LIN {X 0,Y 367.655,Z 436.574,A -85,B 0,C 180,E1 -12880.464,E2 -12880.464} C_VEL
LIN {X 0,Y 367.47,Z 439.697,A -85,B 0,C 180,E1 -12882.738,E2 -12882.738} C_VEL
LIN {X 0,Y 367.357,Z 440.888,A -85,B 0,C 180,E1 -12884.402,E2 -12884.402} C_VEL
LIN {X 0,Y 367.359,Z 441.192,A -85,B 0,C 180,E1 -12885.536,E2 -12885.536} C_VEL
LIN {X 0,Y 367.414,Z 440.944,A -85,B 0,C 180,E1 -12886.98,E2 -12886.98} C_VEL
LIN {X 0,Y 367.622,Z 439.55,A -85,B 0,C 180,E1 -12888.919,E2 -12888.919} C_VEL
LIN {X 0,Y 367.118,Z 438.651,A -85,B 0,C 180,E1 -12889.827,E2 -12889.827} C_VEL
LIN {X 0,Y 364.548,Z 436.647,A -85,B 0,C 180,E1 -12891.296,E2 -12891.296} C_VEL
LIN {X 0,Y 362.068,Z 433.845,A -85,B 0,C 180,E1 -12892.751,E2 -12892.751} C_VEL
LIN {X 0,Y 361.716,Z 431.694,A -85,B 0,C 180,E1 -12893.624,E2 -12893.624} C_VEL
LIN {X 0,Y 362.559,Z 425.865,A -85,B 0,C 180,E1 -12895.55,E2 -12895.55} C_VEL
LIN {X 0,Y 363.427,Z 419.541,A -85,B 0,C 180,E1 -12897.184,E2 -12897.184} C_VEL
LIN {X 0,Y 364.552,Z 411.694,A -85,B 0,C 180,E1 -12898.813,E2 -12898.813} C_VEL
LIN {X 0,Y 365.704,Z 403.264,A -85,B 0,C 180,E1 -12900.234,E2 -12900.234} C_VEL
LIN {X 0,Y 366.982,Z 393.098,A -85,B 0,C 180,E1 -12901.617,E2 -12901.617} C_VEL
LIN {X 0,Y 368.262,Z 382.466,A -85,B 0,C 180,E1 -12902.766,E2 -12902.766} C_VEL
LIN {X 0,Y 369.192,Z 372.107,A -85,B 0,C 180,E1 -12903.67,E2 -12903.67} C_VEL
LIN {X 0,Y 370.135,Z 360.17,A -85,B 0,C 180,E1 -12904.475,E2 -12904.475} C_VEL
LIN {X 0,Y 370.867,Z 347.614,A -85,B 0,C 180,E1 -12905.082,E2 -12905.082} C_VEL
LIN {X 0,Y 371.289,Z 334.414,A -85,B 0,C 180,E1 -12905.493,E2 -12905.493} C_VEL
LIN {X 0,Y 372.995,Z 256.748,A -85,B 0,C 180,E1 -12907.02,E2 -12907.02} C_VEL
LIN {X 0,Y 371.362,Z 249.513,A -85,B 0,C 180,E1 -12907.298,E2 -12907.298} C_VEL
LIN {X 0,Y 364.262,Z 233.198,A -85,B 0,C 180,E1 -12908.217,E2 -12908.217} C_VEL
LIN {X 0,Y 363.464,Z 231.172,A -85,B 0,C 180,E1 -12908.333,E2 -12908.333} C_VEL
LIN {X 0,Y 361.902,Z 224.409,A -85,B 0,C 180,E1 -12910.291,E2 -12910.291} C_VEL
LIN {X 0,Y 361.922,Z 224.406,A -85,B 0,C 180,E1 -12914.35,E2 -12914.35} C_VEL
LIN {X 0,Y 361.875,Z 224.407,A -85,B 0,C 180,E1 -12917.558,E2 -12917.558} C_VEL
LIN {X 0,Y 361.861,Z 224.41,A -85,B 0,C 180,E1 -12920.972,E2 -12920.972} C_VEL
LIN {X 0,Y 361.86,Z 224.405,A -85,B 0,C 180,E1 -12924.654,E2 -12924.654} C_VEL
LIN {X 0,Y 361.822,Z 224.409,A -85,B 0,C 180,E1 -12928.369,E2 -12928.369} C_VEL
LIN {X 0,Y 361.885,Z 224.401,A -85,B 0,C 180,E1 -12930.954,E2 -12930.954} C_VEL
LIN {X 0,Y 361.936,Z 224.399,A -85,B 0,C 180,E1 -12933.474,E2 -12933.474} C_VEL
LIN {X 0,Y 361.884,Z 224.404,A -85,B 0,C 180,E1 -12937.145,E2 -12937.145} C_VEL
LIN {X 0,Y 361.907,Z 224.401,A -85,B 0,C 180,E1 -12940.724,E2 -12940.724} C_VEL
LIN {X 0,Y 361.925,Z 224.4,A -85,B 0,C 180,E1 -12944.226,E2 -12944.226} C_VEL
LIN {X 0,Y 361.977,Z 224.391,A -85,B 0,C 180,E1 -12946.527,E2 -12946.527} C_VEL
LIN {X 0,Y 362.008,Z 224.39,A -85,B 0,C 180,E1 -12949.938,E2 -12949.938} C_VEL
LIN {X 0,Y 362.142,Z 224.371,A -85,B 0,C 180,E1 -12953.314,E2 -12953.314} C_VEL
LIN {X 0,Y 362.254,Z 224.357,A -85,B 0,C 180,E1 -12957.777,E2 -12957.777} C_VEL
LIN {X 0,Y 362.381,Z 224.336,A -85,B 0,C 180,E1 -12960,E2 -12960} C_VEL
LIN {X 0,Y 362.254,Z 224.351,A -85,B 0,C 180,E1 -12962.224,E2 -12962.224} C_VEL
LIN {X 0,Y 362.116,Z 224.367,A -85,B 0,C 180,E1 -12966.688,E2 -12966.688} C_VEL
LIN {X 0,Y 361.98,Z 224.382,A -85,B 0,C 180,E1 -12970.064,E2 -12970.064} C_VEL
LIN {X 0,Y 361.979,Z 224.387,A -85,B 0,C 180,E1 -12973.899,E2 -12973.899} C_VEL
LIN {X 0,Y 361.909,Z 224.405,A -85,B 0,C 180,E1 -12976.936,E2 -12976.936} C_VEL
LIN {X 0,Y 361.856,Z 224.406,A -85,B 0,C 180,E1 -12980.463,E2 -12980.463} C_VEL
LIN {X 0,Y 361.878,Z 224.402,A -85,B 0,C 180,E1 -12984.114,E2 -12984.114} C_VEL
LIN {X 0,Y 361.826,Z 224.408,A -85,B 0,C 180,E1 -12987.786,E2 -12987.786} C_VEL
LIN {X 0,Y 361.812,Z 224.411,A -85,B 0,C 180,E1 -12991.281,E2 -12991.281} C_VEL
LIN {X 0,Y 361.837,Z 224.41,A -85,B 0,C 180,E1 -12994.283,E2 -12994.283} C_VEL
LIN {X 0,Y 361.846,Z 224.407,A -85,B 0,C 180,E1 -12997.223,E2 -12997.223} C_VEL
LIN {X 0,Y 361.82,Z 224.405,A -85,B 0,C 180,E1 -13000.756,E2 -13000.756} C_VEL
LIN {X 0,Y 361.808,Z 224.419,A -85,B 0,C 180,E1 -13004.37,E2 -13004.37} C_VEL
LIN {X 0,Y 361.824,Z 224.413,A -85,B 0,C 180,E1 -13007.571,E2 -13007.571} C_VEL
LIN {X 0,Y 361.838,Z 224.414,A -85,B 0,C 180,E1 -13011.573,E2 -13011.573} C_VEL
LIN {X 0,Y 361.871,Z 224.411,A -85,B 0,C 180,E1 -13014.657,E2 -13014.657} C_VEL
LIN {X 0,Y 361.893,Z 224.531,A -85,B 0,C 180,E1 -13018.009,E2 -13018.009} C_VEL
LIN {X 0,Y 364.748,Z 236.504,A -85,B 0,C 180,E1 -13021.204,E2 -13021.204} C_VEL
LIN {X 0,Y 366.845,Z 247.054,A -85,B 0,C 180,E1 -13023.856,E2 -13023.856} C_VEL
LIN {X 0,Y 365.526,Z 260.284,A -85,B 0,C 180,E1 -13026.786,E2 -13026.786} C_VEL
LIN {X 0,Y 365.523,Z 261.046,A -85,B 0,C 180,E1 -13026.908,E2 -13026.908} C_VEL
LIN {X 0,Y 370.371,Z 285.77,A -85,B 0,C 180,E1 -13027.813,E2 -13027.813} C_VEL
LIN {X 0,Y 372.176,Z 298.437,A -85,B 0,C 180,E1 -13028.214,E2 -13028.214} C_VEL
LIN {X 0,Y 370.738,Z 369.995,A -85,B 0,C 180,E1 -13029.651,E2 -13029.651} C_VEL
LIN {X 0,Y 369.975,Z 383.064,A -85,B 0,C 180,E1 -13030.114,E2 -13030.114} C_VEL
LIN {X 0,Y 368.862,Z 396.243,A -85,B 0,C 180,E1 -13030.812,E2 -13030.812} C_VEL
LIN {X 0,Y 367.742,Z 407.347,A -85,B 0,C 180,E1 -13031.619,E2 -13031.619} C_VEL
LIN {X 0,Y 366.396,Z 418.906,A -85,B 0,C 180,E1 -13032.703,E2 -13032.703} C_VEL
LIN {X 0,Y 365.129,Z 429.333,A -85,B 0,C 180,E1 -13033.937,E2 -13033.937} C_VEL
LIN {X 0,Y 363.957,Z 438.087,A -85,B 0,C 180,E1 -13035.208,E2 -13035.208} C_VEL
LIN {X 0,Y 363.049,Z 445.79,A -85,B 0,C 180,E1 -13036.567,E2 -13036.567} C_VEL
LIN {X 0,Y 361.938,Z 453.565,A -85,B 0,C 180,E1 -13038.235,E2 -13038.235} C_VEL
LIN {X 0,Y 361.235,Z 459.821,A -85,B 0,C 180,E1 -13039.915,E2 -13039.915} C_VEL
LIN {X 0,Y 360.761,Z 464.821,A -85,B 0,C 180,E1 -13041.597,E2 -13041.597} C_VEL
LIN {X 0,Y 360.487,Z 468.707,A -85,B 0,C 180,E1 -13043.281,E2 -13043.281} C_VEL
LIN {X 0,Y 360.362,Z 472.323,A -85,B 0,C 180,E1 -13045.524,E2 -13045.524} C_VEL
LIN {X 0,Y 360.322,Z 473.506,A -85,B 0,C 180,E1 -13046.644,E2 -13046.644} C_VEL
LIN {X 0,Y 360.455,Z 474.626,A -85,B 0,C 180,E1 -13048.881,E2 -13048.881} C_VEL
LIN {X 0,Y 360.48,Z 474.603,A -85,B 0,C 180,E1 -13049.998,E2 -13049.998} C_VEL
LIN {X 0,Y 360.476,Z 474.18,A -85,B 0,C 180,E1 -13051.115,E2 -13051.115} C_VEL
LIN {X 0,Y 360.392,Z 473.312,A -85,B 0,C 180,E1 -13052.233,E2 -13052.233} C_VEL
LIN {X 0,Y 360.437,Z 470.367,A -85,B 0,C 180,E1 -13054.471,E2 -13054.471} C_VEL
LIN {X 0,Y 360.443,Z 467.183,A -85,B 0,C 180,E1 -13056.058,E2 -13056.058} C_VEL
LIN {X 0,Y 360.61,Z 462.477,A -85,B 0,C 180,E1 -13057.838,E2 -13057.838} C_VEL
LIN {X 0,Y 361.014,Z 455.655,A -85,B 0,C 180,E1 -13059.805,E2 -13059.805} C_VEL
LIN {X 0,Y 361.556,Z 448.205,A -85,B 0,C 180,E1 -13061.49,E2 -13061.49} C_VEL
LIN {X 0,Y 362.236,Z 440.615,A -85,B 0,C 180,E1 -13062.889,E2 -13062.889} C_VEL
LIN {X 0,Y 363.097,Z 431.416,A -85,B 0,C 180,E1 -13064.284,E2 -13064.284} C_VEL
LIN {X 0,Y 363.919,Z 421.332,A -85,B 0,C 180,E1 -13065.525,E2 -13065.525} C_VEL
LIN {X 0,Y 364.881,Z 409.851,A -85,B 0,C 180,E1 -13066.645,E2 -13066.645} C_VEL
LIN {X 0,Y 365.786,Z 398.096,A -85,B 0,C 180,E1 -13067.539,E2 -13067.539} C_VEL
LIN {X 0,Y 366.634,Z 385.333,A -85,B 0,C 180,E1 -13068.254,E2 -13068.254} C_VEL
LIN {X 0,Y 367.224,Z 372.882,A -85,B 0,C 180,E1 -13068.729,E2 -13068.729} C_VEL
LIN {X 0,Y 367.62,Z 352.948,A -85,B 0,C 180,E1 -13069.167,E2 -13069.167} C_VEL
LIN {X 0,Y 368.305,Z 295.909,A -85,B 0,C 180,E1 -13070.285,E2 -13070.285} C_VEL
LIN {X 0,Y 363.695,Z 261.588,A -85,B 0,C 180,E1 -13071.209,E2 -13071.209} C_VEL
LIN {X 0,Y 365.183,Z 243.676,A -85,B 0,C 180,E1 -13075.044,E2 -13075.044} C_VEL
LIN {X 0,Y 364.894,Z 239.411,A -85,B 0,C 180,E1 -13075.999,E2 -13075.999} C_VEL
LIN {X 0,Y 362.703,Z 228.105,A -85,B 0,C 180,E1 -13078.652,E2 -13078.652} C_VEL
LIN {X 0,Y 361.913,Z 224.405,A -85,B 0,C 180,E1 -13079.588,E2 -13079.588} C_VEL
LIN {X 0,Y 361.844,Z 224.409,A -85,B 0,C 180,E1 -13083.365,E2 -13083.365} C_VEL
LIN {X 0,Y 361.849,Z 224.408,A -85,B 0,C 180,E1 -13087.014,E2 -13087.014} C_VEL
LIN {X 0,Y 361.834,Z 224.416,A -85,B 0,C 180,E1 -13089.857,E2 -13089.857} C_VEL
LIN {X 0,Y 361.815,Z 224.412,A -85,B 0,C 180,E1 -13092.824,E2 -13092.824} C_VEL
LIN {X 0,Y 361.871,Z 224.411,A -85,B 0,C 180,E1 -13095.93,E2 -13095.93} C_VEL
LIN {X 0,Y 361.879,Z 224.406,A -85,B 0,C 180,E1 -13099.228,E2 -13099.228} C_VEL
LIN {X 0,Y 361.838,Z 224.41,A -85,B 0,C 180,E1 -13102.978,E2 -13102.978} C_VEL
LIN {X 0,Y 361.825,Z 224.411,A -85,B 0,C 180,E1 -13106.627,E2 -13106.627} C_VEL
LIN {X 0,Y 361.841,Z 224.415,A -85,B 0,C 180,E1 -13109.669,E2 -13109.669} C_VEL
LIN {X 0,Y 361.917,Z 224.405,A -85,B 0,C 180,E1 -13113.472,E2 -13113.472} C_VEL
LIN {X 0,Y 361.875,Z 224.408,A -85,B 0,C 180,E1 -13117.143,E2 -13117.143} C_VEL
LIN {X 0,Y 361.891,Z 224.403,A -85,B 0,C 180,E1 -13120.722,E2 -13120.722} C_VEL
LIN {X 0,Y 361.904,Z 224.401,A -85,B 0,C 180,E1 -13124.224,E2 -13124.224} C_VEL
LIN {X 0,Y 361.956,Z 224.395,A -85,B 0,C 180,E1 -13126.526,E2 -13126.526} C_VEL
LIN {X 0,Y 361.992,Z 224.391,A -85,B 0,C 180,E1 -13129.937,E2 -13129.937} C_VEL
LIN {X 0,Y 362.112,Z 224.375,A -85,B 0,C 180,E1 -13132.191,E2 -13132.191} C_VEL
LIN {X 0,Y 362.08,Z 224.38,A -85,B 0,C 180,E1 -13134.43,E2 -13134.43} C_VEL
LIN {X 0,Y 362.234,Z 224.361,A -85,B 0,C 180,E1 -13137.776,E2 -13137.776} C_VEL
LIN {X 0,Y 362.38,Z 224.342,A -85,B 0,C 180,E1 -13140,E2 -13140} C_VEL
LIN {X 0,Y 362.231,Z 224.361,A -85,B 0,C 180,E1 -13142.224,E2 -13142.224} C_VEL
LIN {X 0,Y 362.111,Z 224.379,A -85,B 0,C 180,E1 -13146.687,E2 -13146.687} C_VEL
LIN {X 0,Y 361.987,Z 224.391,A -85,B 0,C 180,E1 -13150.063,E2 -13150.063} C_VEL
LIN {X 0,Y 361.954,Z 224.395,A -85,B 0,C 180,E1 -13153.9,E2 -13153.9} C_VEL
LIN {X 0,Y 361.91,Z 224.4,A -85,B 0,C 180,E1 -13157.933,E2 -13157.933} C_VEL
LIN {X 0,Y 361.819,Z 224.412,A -85,B 0,C 180,E1 -13161.657,E2 -13161.657} C_VEL
LIN {X 0,Y 361.886,Z 224.404,A -85,B 0,C 180,E1 -13165.293,E2 -13165.293} C_VEL
LIN {X 0,Y 361.867,Z 224.406,A -85,B 0,C 180,E1 -13167.782,E2 -13167.782} C_VEL
LIN {X 0,Y 361.797,Z 224.415,A -85,B 0,C 180,E1 -13171.633,E2 -13171.633} C_VEL
LIN {X 0,Y 361.839,Z 224.409,A -85,B 0,C 180,E1 -13175.348,E2 -13175.348} C_VEL
LIN {X 0,Y 361.832,Z 224.411,A -85,B 0,C 180,E1 -13179.029,E2 -13179.029} C_VEL
LIN {X 0,Y 361.806,Z 224.415,A -85,B 0,C 180,E1 -13182.833,E2 -13182.833} C_VEL
LIN {X 0,Y 361.79,Z 224.418,A -85,B 0,C 180,E1 -13185.951,E2 -13185.951} C_VEL
LIN {X 0,Y 361.81,Z 224.413,A -85,B 0,C 180,E1 -13189.249,E2 -13189.249} C_VEL
LIN {X 0,Y 361.842,Z 224.41,A -85,B 0,C 180,E1 -13192.781,E2 -13192.781} C_VEL
LIN {X 0,Y 361.835,Z 224.412,A -85,B 0,C 180,E1 -13195.723,E2 -13195.723} C_VEL
LIN {X 0,Y 361.856,Z 224.41,A -85,B 0,C 180,E1 -13199.676,E2 -13199.676} C_VEL
LIN {X 0,Y 361.94,Z 224.398,A -85,B 0,C 180,E1 -13203.479,E2 -13203.479} C_VEL
LIN {X 0,Y 361.868,Z 224.406,A -85,B 0,C 180,E1 -13207.148,E2 -13207.148} C_VEL
LIN {X 0,Y 361.876,Z 224.405,A -85,B 0,C 180,E1 -13210.726,E2 -13210.726} C_VEL
LIN {X 0,Y 361.936,Z 224.399,A -85,B 0,C 180,E1 -13214.229,E2 -13214.229} C_VEL
LIN {X 0,Y 361.993,Z 224.39,A -85,B 0,C 180,E1 -13216.531,E2 -13216.531} C_VEL
LIN {X 0,Y 362.023,Z 224.39,A -85,B 0,C 180,E1 -13219.941,E2 -13219.941} C_VEL
LIN {X 0,Y 362.107,Z 224.517,A -85,B 0,C 180,E1 -13222.299,E2 -13222.299} C_VEL
LIN {X 0,Y 363.257,Z 230.458,A -85,B 0,C 180,E1 -13223.854,E2 -13223.854} C_VEL
LIN {X 0,Y 366.565,Z 241.792,A -85,B 0,C 180,E1 -13224.261,E2 -13224.261} C_VEL
LIN {X 0,Y 368.991,Z 255.095,A -85,B 0,C 180,E1 -13224.647,E2 -13224.647} C_VEL
LIN {X 0,Y 367.566,Z 337.574,A -85,B 0,C 180,E1 -13226.268,E2 -13226.268} C_VEL
LIN {X 0,Y 367.149,Z 350.787,A -85,B 0,C 180,E1 -13226.744,E2 -13226.744} C_VEL
LIN {X 0,Y 366.529,Z 364.039,A -85,B 0,C 180,E1 -13227.461,E2 -13227.461} C_VEL
LIN {X 0,Y 365.84,Z 375.392,A -85,B 0,C 180,E1 -13228.3,E2 -13228.3} C_VEL
LIN {X 0,Y 364.88,Z 387.428,A -85,B 0,C 180,E1 -13229.45,E2 -13229.45} C_VEL
LIN {X 0,Y 364.003,Z 397.741,A -85,B 0,C 180,E1 -13230.693,E2 -13230.693} C_VEL
LIN {X 0,Y 363.212,Z 406.181,A -85,B 0,C 180,E1 -13231.942,E2 -13231.942} C_VEL
LIN {X 0,Y 362.346,Z 415.323,A -85,B 0,C 180,E1 -13233.616,E2 -13233.616} C_VEL
LIN {X 0,Y 361.653,Z 422.693,A -85,B 0,C 180,E1 -13235.298,E2 -13235.298} C_VEL
LIN {X 0,Y 361.228,Z 429.07,A -85,B 0,C 180,E1 -13237.142,E2 -13237.142} C_VEL
LIN {X 0,Y 360.799,Z 433.899,A -85,B 0,C 180,E1 -13238.966,E2 -13238.966} C_VEL
LIN {X 0,Y 360.596,Z 436.264,A -85,B 0,C 180,E1 -13240.104,E2 -13240.104} C_VEL
LIN {X 0,Y 360.476,Z 438.192,A -85,B 0,C 180,E1 -13241.244,E2 -13241.244} C_VEL
LIN {X 0,Y 360.384,Z 440.087,A -85,B 0,C 180,E1 -13242.822,E2 -13242.822} C_VEL
LIN {X 0,Y 360.267,Z 441.32,A -85,B 0,C 180,E1 -13244.691,E2 -13244.691} C_VEL
LIN {X 0,Y 360.28,Z 441.54,A -85,B 0,C 180,E1 -13245.849,E2 -13245.849} C_VEL
LIN {X 0,Y 360.354,Z 441.256,A -85,B 0,C 180,E1 -13247.129,E2 -13247.129} C_VEL
LIN {X 0,Y 360.604,Z 439.605,A -85,B 0,C 180,E1 -13249.349,E2 -13249.349} C_VEL
LIN {X 0,Y 360.936,Z 437.572,A -85,B 0,C 180,E1 -13250.831,E2 -13250.831} C_VEL
LIN {X 0,Y 361.455,Z 433.569,A -85,B 0,C 180,E1 -13252.884,E2 -13252.884} C_VEL
LIN {X 0,Y 361.716,Z 431.694,A -85,B 0,C 180,E1 -13253.624,E2 -13253.624} C_VEL
LIN {X 0,Y 361.417,Z 429.409,A -85,B 0,C 180,E1 -13254.486,E2 -13254.486} C_VEL
LIN {X 0,Y 359.236,Z 425.398,A -85,B 0,C 180,E1 -13255.891,E2 -13255.891} C_VEL
LIN {X 0,Y 357.143,Z 420.795,A -85,B 0,C 180,E1 -13257.257,E2 -13257.257} C_VEL
LIN {X 0,Y 356.974,Z 417.487,A -85,B 0,C 180,E1 -13258.043,E2 -13258.043} C_VEL
LIN {X 0,Y 358.231,Z 409.109,A -85,B 0,C 180,E1 -13259.686,E2 -13259.686} C_VEL
LIN {X 0,Y 359.508,Z 399.56,A -85,B 0,C 180,E1 -13261.2,E2 -13261.2} C_VEL
LIN {X 0,Y 360.897,Z 388.88,A -85,B 0,C 180,E1 -13262.544,E2 -13262.544} C_VEL
LIN {X 0,Y 362.179,Z 377.798,A -85,B 0,C 180,E1 -13263.645,E2 -13263.645} C_VEL
LIN {X 0,Y 363.227,Z 366.193,A -85,B 0,C 180,E1 -13264.551,E2 -13264.551} C_VEL
LIN {X 0,Y 364.015,Z 354.796,A -85,B 0,C 180,E1 -13265.224,E2 -13265.224} C_VEL
LIN {X 0,Y 364.622,Z 342.007,A -85,B 0,C 180,E1 -13265.748,E2 -13265.748} C_VEL
LIN {X 0,Y 365.053,Z 324.151,A -85,B 0,C 180,E1 -13266.169,E2 -13266.169} C_VEL
LIN {X 0,Y 366.606,Z 257.171,A -85,B 0,C 180,E1 -13267.503,E2 -13267.503} C_VEL
LIN {X 0,Y 365.006,Z 251.438,A -85,B 0,C 180,E1 -13267.755,E2 -13267.755} C_VEL
LIN {X 0,Y 357.56,Z 234.337,A -85,B 0,C 180,E1 -13268.752,E2 -13268.752} C_VEL
LIN {X 0,Y 356.337,Z 231.522,A -85,B 0,C 180,E1 -13268.929,E2 -13268.929} C_VEL
LIN {X 0,Y 354.871,Z 225.278,A -85,B 0,C 180,E1 -13270.807,E2 -13270.807} C_VEL
LIN {X 0,Y 354.877,Z 225.285,A -85,B 0,C 180,E1 -13274.525,E2 -13274.525} C_VEL
LIN {X 0,Y 354.829,Z 225.284,A -85,B 0,C 180,E1 -13277.668,E2 -13277.668} C_VEL
LIN {X 0,Y 354.81,Z 225.289,A -85,B 0,C 180,E1 -13280.666,E2 -13280.666} C_VEL
LIN {X 0,Y 354.808,Z 225.286,A -85,B 0,C 180,E1 -13284.3,E2 -13284.3} C_VEL
LIN {X 0,Y 354.771,Z 225.29,A -85,B 0,C 180,E1 -13287.665,E2 -13287.665} C_VEL
LIN {X 0,Y 354.854,Z 225.277,A -85,B 0,C 180,E1 -13290.62,E2 -13290.62} C_VEL
LIN {X 0,Y 354.881,Z 225.273,A -85,B 0,C 180,E1 -13294.172,E2 -13294.172} C_VEL
LIN {X 0,Y 354.826,Z 225.281,A -85,B 0,C 180,E1 -13297.894,E2 -13297.894} C_VEL
LIN {X 0,Y 354.905,Z 225.272,A -85,B 0,C 180,E1 -13301.891,E2 -13301.891} C_VEL
LIN {X 0,Y 354.922,Z 225.272,A -85,B 0,C 180,E1 -13305.982,E2 -13305.982} C_VEL
LIN {X 0,Y 354.955,Z 225.27,A -85,B 0,C 180,E1 -13309.736,E2 -13309.736} C_VEL
LIN {X 0,Y 355.105,Z 225.246,A -85,B 0,C 180,E1 -13313.181,E2 -13313.181} C_VEL
LIN {X 0,Y 355.218,Z 225.233,A -85,B 0,C 180,E1 -13317.733,E2 -13317.733} C_VEL
LIN {X 0,Y 355.331,Z 225.214,A -85,B 0,C 180,E1 -13320,E2 -13320} C_VEL
LIN {X 0,Y 355.217,Z 225.228,A -85,B 0,C 180,E1 -13322.268,E2 -13322.268} C_VEL
LIN {X 0,Y 355.081,Z 225.244,A -85,B 0,C 180,E1 -13326.821,E2 -13326.821} C_VEL
LIN {X 0,Y 354.937,Z 225.259,A -85,B 0,C 180,E1 -13330.266,E2 -13330.266} C_VEL
LIN {X 0,Y 354.923,Z 225.265,A -85,B 0,C 180,E1 -13334.019,E2 -13334.019} C_VEL
LIN {X 0,Y 354.86,Z 225.279,A -85,B 0,C 180,E1 -13337.282,E2 -13337.282} C_VEL
LIN {X 0,Y 354.8,Z 225.287,A -85,B 0,C 180,E1 -13341.418,E2 -13341.418} C_VEL
LIN {X 0,Y 354.833,Z 225.283,A -85,B 0,C 180,E1 -13344.579,E2 -13344.579} C_VEL
LIN {X 0,Y 354.785,Z 225.288,A -85,B 0,C 180,E1 -13348.387,E2 -13348.387} C_VEL
LIN {X 0,Y 354.766,Z 225.293,A -85,B 0,C 180,E1 -13352.336,E2 -13352.336} C_VEL
LIN {X 0,Y 354.806,Z 225.287,A -85,B 0,C 180,E1 -13355.7,E2 -13355.7} C_VEL
LIN {X 0,Y 354.79,Z 225.29,A -85,B 0,C 180,E1 -13359.42,E2 -13359.42} C_VEL
LIN {X 0,Y 354.777,Z 225.284,A -85,B 0,C 180,E1 -13362.868,E2 -13362.868} C_VEL
LIN {X 0,Y 354.758,Z 225.295,A -85,B 0,C 180,E1 -13366.105,E2 -13366.105} C_VEL
LIN {X 0,Y 354.76,Z 225.292,A -85,B 0,C 180,E1 -13369.177,E2 -13369.177} C_VEL
LIN {X 0,Y 354.796,Z 225.287,A -85,B 0,C 180,E1 -13372.406,E2 -13372.406} C_VEL
LIN {X 0,Y 354.809,Z 225.29,A -85,B 0,C 180,E1 -13374.942,E2 -13374.942} C_VEL
LIN {X 0,Y 354.826,Z 225.448,A -85,B 0,C 180,E1 -13377.504,E2 -13377.504} C_VEL
LIN {X 0,Y 357.59,Z 236.589,A -85,B 0,C 180,E1 -13380.572,E2 -13380.572} C_VEL
LIN {X 0,Y 359.751,Z 247.108,A -85,B 0,C 180,E1 -13383.3,E2 -13383.3} C_VEL
LIN {X 0,Y 359.891,Z 250.492,A -85,B 0,C 180,E1 -13384.111,E2 -13384.111} C_VEL
LIN {X 0,Y 358.807,Z 260.39,A -85,B 0,C 180,E1 -13386.34,E2 -13386.34} C_VEL
LIN {X 0,Y 364.007,Z 286.877,A -85,B 0,C 180,E1 -13387.353,E2 -13387.353} C_VEL
LIN {X 0,Y 365.72,Z 299.035,A -85,B 0,C 180,E1 -13387.749,E2 -13387.749} C_VEL
LIN {X 0,Y 364.264,Z 369.785,A -85,B 0,C 180,E1 -13389.199,E2 -13389.199} C_VEL
LIN {X 0,Y 363.42,Z 383.567,A -85,B 0,C 180,E1 -13389.703,E2 -13389.703} C_VEL
LIN {X 0,Y 362.31,Z 395.969,A -85,B 0,C 180,E1 -13390.377,E2 -13390.377} C_VEL
LIN {X 0,Y 361.04,Z 407.844,A -85,B 0,C 180,E1 -13391.265,E2 -13391.265} C_VEL
LIN {X 0,Y 359.647,Z 419.252,A -85,B 0,C 180,E1 -13392.368,E2 -13392.368} C_VEL
LIN {X 0,Y 358.304,Z 429.563,A -85,B 0,C 180,E1 -13393.622,E2 -13393.622} C_VEL
LIN {X 0,Y 356.891,Z 439.678,A -85,B 0,C 180,E1 -13395.167,E2 -13395.167} C_VEL
LIN {X 0,Y 355.701,Z 448.575,A -85,B 0,C 180,E1 -13396.866,E2 -13396.866} C_VEL
LIN {X 0,Y 354.647,Z 455.761,A -85,B 0,C 180,E1 -13398.569,E2 -13398.569} C_VEL
LIN {X 0,Y 354.013,Z 461.523,A -85,B 0,C 180,E1 -13400.284,E2 -13400.284} C_VEL
LIN {X 0,Y 353.573,Z 466.087,A -85,B 0,C 180,E1 -13402.001,E2 -13402.001} C_VEL
LIN {X 0,Y 353.316,Z 470.087,A -85,B 0,C 180,E1 -13404.033,E2 -13404.033} C_VEL
LIN {X 0,Y 353.274,Z 472.081,A -85,B 0,C 180,E1 -13405.434,E2 -13405.434} C_VEL
LIN {X 0,Y 353.242,Z 473.226,A -85,B 0,C 180,E1 -13406.576,E2 -13406.576} C_VEL
LIN {X 0,Y 353.357,Z 474.307,A -85,B 0,C 180,E1 -13408.858,E2 -13408.858} C_VEL
LIN {X 0,Y 353.399,Z 474.266,A -85,B 0,C 180,E1 -13409.998,E2 -13409.998} C_VEL
LIN {X 0,Y 353.394,Z 473.808,A -85,B 0,C 180,E1 -13411.137,E2 -13411.137} C_VEL
LIN {X 0,Y 353.265,Z 471.626,A -85,B 0,C 180,E1 -13413.419,E2 -13413.419} C_VEL
LIN {X 0,Y 353.32,Z 468.879,A -85,B 0,C 180,E1 -13415.133,E2 -13415.133} C_VEL
LIN {X 0,Y 353.415,Z 465.087,A -85,B 0,C 180,E1 -13416.85,E2 -13416.85} C_VEL
LIN {X 0,Y 353.639,Z 460.15,A -85,B 0,C 180,E1 -13418.569,E2 -13418.569} C_VEL
LIN {X 0,Y 354.036,Z 453.919,A -85,B 0,C 180,E1 -13420.289,E2 -13420.289} C_VEL
LIN {X 0,Y 354.713,Z 446.152,A -85,B 0,C 180,E1 -13422.004,E2 -13422.004} C_VEL
LIN {X 0,Y 355.626,Z 436.381,A -85,B 0,C 180,E1 -13423.715,E2 -13423.715} C_VEL
LIN {X 0,Y 356.496,Z 426.492,A -85,B 0,C 180,E1 -13425.109,E2 -13425.109} C_VEL
LIN {X 0,Y 357.332,Z 416.24,A -85,B 0,C 180,E1 -13426.273,E2 -13426.273} C_VEL
LIN {X 0,Y 358.323,Z 405.353,A -85,B 0,C 180,E1 -13427.253,E2 -13427.253} C_VEL
LIN {X 0,Y 359.3,Z 392.207,A -85,B 0,C 180,E1 -13428.16,E2 -13428.16} C_VEL
LIN {X 0,Y 360.042,Z 379.413,A -85,B 0,C 180,E1 -13428.785,E2 -13428.785} C_VEL
LIN {X 0,Y 360.576,Z 365.93,A -85,B 0,C 180,E1 -13429.199,E2 -13429.199} C_VEL
LIN {X 0,Y 361.476,Z 296.542,A -85,B 0,C 180,E1 -13430.588,E2 -13430.588} C_VEL
LIN {X 0,Y 356.75,Z 261.283,A -85,B 0,C 180,E1 -13431.557,E2 -13431.557} C_VEL
LIN {X 0,Y 358.12,Z 245.721,A -85,B 0,C 180,E1 -13434.952,E2 -13434.952} C_VEL
LIN {X 0,Y 358.074,Z 241.554,A -85,B 0,C 180,E1 -13435.889,E2 -13435.889} C_VEL
LIN {X 0,Y 355.896,Z 230.166,A -85,B 0,C 180,E1 -13438.606,E2 -13438.606} C_VEL
LIN {X 0,Y 354.839,Z 225.287,A -85,B 0,C 180,E1 -13439.838,E2 -13439.838} C_VEL
LIN {X 0,Y 354.792,Z 225.29,A -85,B 0,C 180,E1 -13443.698,E2 -13443.698} C_VEL
LIN {X 0,Y 354.78,Z 225.29,A -85,B 0,C 180,E1 -13446.455,E2 -13446.455} C_VEL
LIN {X 0,Y 354.805,Z 225.287,A -85,B 0,C 180,E1 -13449.419,E2 -13449.419} C_VEL
LIN {X 0,Y 354.767,Z 225.29,A -85,B 0,C 180,E1 -13452.863,E2 -13452.863} C_VEL
LIN {X 0,Y 354.814,Z 225.288,A -85,B 0,C 180,E1 -13456.11,E2 -13456.11} C_VEL
LIN {X 0,Y 354.83,Z 225.283,A -85,B 0,C 180,E1 -13459.184,E2 -13459.184} C_VEL
LIN {X 0,Y 354.779,Z 225.289,A -85,B 0,C 180,E1 -13462.398,E2 -13462.398} C_VEL
LIN {X 0,Y 354.78,Z 225.289,A -85,B 0,C 180,E1 -13464.937,E2 -13464.937} C_VEL
LIN {X 0,Y 354.759,Z 225.291,A -85,B 0,C 180,E1 -13468.402,E2 -13468.402} C_VEL
LIN {X 0,Y 354.815,Z 225.29,A -85,B 0,C 180,E1 -13471.616,E2 -13471.616} C_VEL
LIN {X 0,Y 354.862,Z 225.279,A -85,B 0,C 180,E1 -13474.169,E2 -13474.169} C_VEL
LIN {X 0,Y 354.818,Z 225.286,A -85,B 0,C 180,E1 -13477.892,E2 -13477.892} C_VEL
LIN {X 0,Y 354.883,Z 225.277,A -85,B 0,C 180,E1 -13481.889,E2 -13481.889} C_VEL
LIN {X 0,Y 354.9,Z 225.274,A -85,B 0,C 180,E1 -13485.98,E2 -13485.98} C_VEL
LIN {X 0,Y 354.939,Z 225.271,A -85,B 0,C 180,E1 -13489.734,E2 -13489.734} C_VEL
LIN {X 0,Y 355.072,Z 225.252,A -85,B 0,C 180,E1 -13492.036,E2 -13492.036} C_VEL
LIN {X 0,Y 355.055,Z 225.254,A -85,B 0,C 180,E1 -13494.32,E2 -13494.32} C_VEL
LIN {X 0,Y 355.197,Z 225.238,A -85,B 0,C 180,E1 -13497.732,E2 -13497.732} C_VEL
LIN {X 0,Y 355.329,Z 225.22,A -85,B 0,C 180,E1 -13500,E2 -13500} C_VEL
LIN {X 0,Y 355.194,Z 225.237,A -85,B 0,C 180,E1 -13502.268,E2 -13502.268} C_VEL
LIN {X 0,Y 355.075,Z 225.257,A -85,B 0,C 180,E1 -13506.82,E2 -13506.82} C_VEL
LIN {X 0,Y 354.934,Z 225.27,A -85,B 0,C 180,E1 -13510.265,E2 -13510.265} C_VEL
LIN {X 0,Y 354.899,Z 225.274,A -85,B 0,C 180,E1 -13514.019,E2 -13514.019} C_VEL
LIN {X 0,Y 354.869,Z 225.278,A -85,B 0,C 180,E1 -13518.104,E2 -13518.104} C_VEL
LIN {X 0,Y 354.773,Z 225.29,A -85,B 0,C 180,E1 -13522.11,E2 -13522.11} C_VEL
LIN {X 0,Y 354.858,Z 225.279,A -85,B 0,C 180,E1 -13525.83,E2 -13525.83} C_VEL
LIN {X 0,Y 354.764,Z 225.291,A -85,B 0,C 180,E1 -13529.686,E2 -13529.686} C_VEL
LIN {X 0,Y 354.78,Z 225.289,A -85,B 0,C 180,E1 -13533.687,E2 -13533.687} C_VEL
LIN {X 0,Y 354.763,Z 225.297,A -85,B 0,C 180,E1 -13536.463,E2 -13536.463} C_VEL
LIN {X 0,Y 354.794,Z 225.287,A -85,B 0,C 180,E1 -13539.427,E2 -13539.427} C_VEL
LIN {X 0,Y 354.758,Z 225.293,A -85,B 0,C 180,E1 -13542.871,E2 -13542.871} C_VEL
LIN {X 0,Y 354.739,Z 225.298,A -85,B 0,C 180,E1 -13546.107,E2 -13546.107} C_VEL
LIN {X 0,Y 354.763,Z 225.291,A -85,B 0,C 180,E1 -13549.183,E2 -13549.183} C_VEL
LIN {X 0,Y 354.785,Z 225.292,A -85,B 0,C 180,E1 -13552.407,E2 -13552.407} C_VEL
LIN {X 0,Y 354.792,Z 225.287,A -85,B 0,C 180,E1 -13554.945,E2 -13554.945} C_VEL
LIN {X 0,Y 354.776,Z 225.292,A -85,B 0,C 180,E1 -13558.409,E2 -13558.409} C_VEL
LIN {X 0,Y 354.831,Z 225.285,A -85,B 0,C 180,E1 -13561.622,E2 -13561.622} C_VEL
LIN {X 0,Y 354.885,Z 225.28,A -85,B 0,C 180,E1 -13564.176,E2 -13564.176} C_VEL
LIN {X 0,Y 354.804,Z 225.292,A -85,B 0,C 180,E1 -13567.896,E2 -13567.896} C_VEL
LIN {X 0,Y 354.881,Z 225.282,A -85,B 0,C 180,E1 -13571.911,E2 -13571.911} C_VEL
LIN {X 0,Y 354.937,Z 225.273,A -85,B 0,C 180,E1 -13575.984,E2 -13575.984} C_VEL
LIN {X 0,Y 354.971,Z 225.271,A -85,B 0,C 180,E1 -13579.739,E2 -13579.739} C_VEL
LIN {X 0,Y 355.056,Z 225.312,A -85,B 0,C 180,E1 -13582.038,E2 -13582.038} C_VEL
LIN {X 0,Y 356.182,Z 231.032,A -85,B 0,C 180,E1 -13583.513,E2 -13583.513} C_VEL
LIN {X 0,Y 359.974,Z 243.656,A -85,B 0,C 180,E1 -13583.971,E2 -13583.971} C_VEL
LIN {X 0,Y 362.217,Z 255.087,A -85,B 0,C 180,E1 -13584.32,E2 -13584.32} C_VEL
LIN {X 0,Y 360.718,Z 338.248,A -85,B 0,C 180,E1 -13585.987,E2 -13585.987} C_VEL
LIN {X 0,Y 360.288,Z 351.342,A -85,B 0,C 180,E1 -13586.472,E2 -13586.472} C_VEL
LIN {X 0,Y 359.7,Z 363.422,A -85,B 0,C 180,E1 -13587.132,E2 -13587.132} C_VEL
LIN {X 0,Y 358.995,Z 375.393,A -85,B 0,C 180,E1 -13588.018,E2 -13588.018} C_VEL
LIN {X 0,Y 358.006,Z 387.216,A -85,B 0,C 180,E1 -13589.158,E2 -13589.158} C_VEL
LIN {X 0,Y 357.093,Z 397.626,A -85,B 0,C 180,E1 -13590.425,E2 -13590.425} C_VEL
LIN {X 0,Y 356.267,Z 406.149,A -85,B 0,C 180,E1 -13591.697,E2 -13591.697} C_VEL
LIN {X 0,Y 355.465,Z 414.011,A -85,B 0,C 180,E1 -13593.118,E2 -13593.118} C_VEL
LIN {X 0,Y 354.772,Z 421.668,A -85,B 0,C 180,E1 -13594.831,E2 -13594.831} C_VEL
LIN {X 0,Y 354.215,Z 428.733,A -85,B 0,C 180,E1 -13596.838,E2 -13596.838} C_VEL
LIN {X 0,Y 353.789,Z 433.44,A -85,B 0,C 180,E1 -13598.569,E2 -13598.569} C_VEL
LIN {X 0,Y 353.472,Z 437.031,A -85,B 0,C 180,E1 -13600.309,E2 -13600.309} C_VEL
LIN {X 0,Y 353.383,Z 438.84,A -85,B 0,C 180,E1 -13601.472,E2 -13601.472} C_VEL
LIN {X 0,Y 353.275,Z 440.461,A -85,B 0,C 180,E1 -13602.892,E2 -13602.892} C_VEL
LIN {X 0,Y 353.182,Z 441.739,A -85,B 0,C 180,E1 -13604.993,E2 -13604.993} C_VEL
LIN {X 0,Y 353.289,Z 441.57,A -85,B 0,C 180,E1 -13607.281,E2 -13607.281} C_VEL
LIN {X 0,Y 353.428,Z 440.829,A -85,B 0,C 180,E1 -13608.552,E2 -13608.552} C_VEL
LIN {X 0,Y 353.601,Z 439.65,A -85,B 0,C 180,E1 -13609.748,E2 -13609.748} C_VEL
LIN {X 0,Y 353.897,Z 437.883,A -85,B 0,C 180,E1 -13611.035,E2 -13611.035} C_VEL
LIN {X 0,Y 354.349,Z 434.683,A -85,B 0,C 180,E1 -13612.753,E2 -13612.753} C_VEL
LIN {X 0,Y 355.032,Z 430.16,A -85,B 0,C 180,E1 -13614.563,E2 -13614.563} C_VEL
LIN {X 0,Y 355.96,Z 424.306,A -85,B 0,C 180,E1 -13616.374,E2 -13616.374} C_VEL
LIN {X 0,Y 356.974,Z 417.487,A -85,B 0,C 180,E1 -13618.043,E2 -13618.043} C_VEL
LIN {X 0,Y 356.851,Z 414.027,A -85,B 0,C 180,E1 -13618.807,E2 -13618.807} C_VEL
LIN {X 0,Y 355.012,Z 408.163,A -85,B 0,C 180,E1 -13620.068,E2 -13620.068} C_VEL
LIN {X 0,Y 353.238,Z 401.838,A -85,B 0,C 180,E1 -13621.266,E2 -13621.266} C_VEL
LIN {X 0,Y 353.2,Z 397.537,A -85,B 0,C 180,E1 -13621.92,E2 -13621.92} C_VEL
LIN {X 0,Y 354.606,Z 387.087,A -85,B 0,C 180,E1 -13623.195,E2 -13623.195} C_VEL
LIN {X 0,Y 355.829,Z 376.149,A -85,B 0,C 180,E1 -13624.263,E2 -13624.263} C_VEL
LIN {X 0,Y 356.898,Z 364.108,A -85,B 0,C 180,E1 -13625.168,E2 -13625.168} C_VEL
LIN {X 0,Y 357.806,Z 350.965,A -85,B 0,C 180,E1 -13625.886,E2 -13625.886} C_VEL
LIN {X 0,Y 358.338,Z 338.23,A -85,B 0,C 180,E1 -13626.349,E2 -13626.349} C_VEL
LIN {X 0,Y 360.207,Z 258.21,A -85,B 0,C 180,E1 -13627.995,E2 -13627.995} C_VEL
LIN {X 0,Y 359.031,Z 254.207,A -85,B 0,C 180,E1 -13628.182,E2 -13628.182} C_VEL
LIN {X 0,Y 351.727,Z 237.443,A -85,B 0,C 180,E1 -13629.192,E2 -13629.192} C_VEL
LIN {X 0,Y 349.168,Z 231.869,A -85,B 0,C 180,E1 -13629.569,E2 -13629.569} C_VEL
LIN {X 0,Y 347.791,Z 226.157,A -85,B 0,C 180,E1 -13631.332,E2 -13631.332} C_VEL
LIN {X 0,Y 347.821,Z 226.161,A -85,B 0,C 180,E1 -13635.005,E2 -13635.005} C_VEL
LIN {X 0,Y 347.774,Z 226.166,A -85,B 0,C 180,E1 -13638.39,E2 -13638.39} C_VEL
LIN {X 0,Y 347.762,Z 226.164,A -85,B 0,C 180,E1 -13642.01,E2 -13642.01} C_VEL
LIN {X 0,Y 347.73,Z 226.164,A -85,B 0,C 180,E1 -13645.535,E2 -13645.535} C_VEL
LIN {X 0,Y 347.749,Z 226.166,A -85,B 0,C 180,E1 -13649.652,E2 -13649.652} C_VEL
LIN {X 0,Y 347.836,Z 226.153,A -85,B 0,C 180,E1 -13652.744,E2 -13652.744} C_VEL
LIN {X 0,Y 347.776,Z 226.162,A -85,B 0,C 180,E1 -13656.161,E2 -13656.161} C_VEL
LIN {X 0,Y 347.809,Z 226.156,A -85,B 0,C 180,E1 -13659.909,E2 -13659.909} C_VEL
LIN {X 0,Y 347.847,Z 226.148,A -85,B 0,C 180,E1 -13662.359,E2 -13662.359} C_VEL
LIN {X 0,Y 347.879,Z 226.149,A -85,B 0,C 180,E1 -13665.97,E2 -13665.97} C_VEL
LIN {X 0,Y 347.906,Z 226.151,A -85,B 0,C 180,E1 -13669.525,E2 -13669.525} C_VEL
LIN {X 0,Y 348.071,Z 226.12,A -85,B 0,C 180,E1 -13673.042,E2 -13673.042} C_VEL
LIN {X 0,Y 348.18,Z 226.109,A -85,B 0,C 180,E1 -13677.687,E2 -13677.687} C_VEL
LIN {X 0,Y 348.282,Z 226.092,A -85,B 0,C 180,E1 -13680,E2 -13680} C_VEL
LIN {X 0,Y 348.18,Z 226.104,A -85,B 0,C 180,E1 -13682.314,E2 -13682.314} C_VEL
LIN {X 0,Y 348.049,Z 226.121,A -85,B 0,C 180,E1 -13686.959,E2 -13686.959} C_VEL
LIN {X 0,Y 347.877,Z 226.138,A -85,B 0,C 180,E1 -13690.476,E2 -13690.476} C_VEL
LIN {X 0,Y 347.881,Z 226.143,A -85,B 0,C 180,E1 -13694.151,E2 -13694.151} C_VEL
LIN {X 0,Y 347.812,Z 226.155,A -85,B 0,C 180,E1 -13697.644,E2 -13697.644} C_VEL
LIN {X 0,Y 347.749,Z 226.165,A -85,B 0,C 180,E1 -13701.626,E2 -13701.626} C_VEL
LIN {X 0,Y 347.752,Z 226.168,A -85,B 0,C 180,E1 -13705.113,E2 -13705.113} C_VEL
LIN {X 0,Y 347.72,Z 226.165,A -85,B 0,C 180,E1 -13707.702,E2 -13707.702} C_VEL
LIN {X 0,Y 347.715,Z 226.17,A -85,B 0,C 180,E1 -13710.352,E2 -13710.352} C_VEL
LIN {X 0,Y 347.736,Z 226.167,A -85,B 0,C 180,E1 -13714.045,E2 -13714.045} C_VEL
LIN {X 0,Y 347.744,Z 226.163,A -85,B 0,C 180,E1 -13717.323,E2 -13717.323} C_VEL
LIN {X 0,Y 347.71,Z 226.167,A -85,B 0,C 180,E1 -13720.301,E2 -13720.301} C_VEL
LIN {X 0,Y 347.715,Z 226.17,A -85,B 0,C 180,E1 -13723.41,E2 -13723.41} C_VEL
LIN {X 0,Y 347.718,Z 226.172,A -85,B 0,C 180,E1 -13726.688,E2 -13726.688} C_VEL
LIN {X 0,Y 347.697,Z 226.167,A -85,B 0,C 180,E1 -13730.184,E2 -13730.184} C_VEL
LIN {X 0,Y 347.752,Z 226.163,A -85,B 0,C 180,E1 -13732.68,E2 -13732.68} C_VEL
LIN {X 0,Y 347.747,Z 226.165,A -85,B 0,C 180,E1 -13735.957,E2 -13735.957} C_VEL
LIN {X 0,Y 347.79,Z 226.227,A -85,B 0,C 180,E1 -13736.935,E2 -13736.935} C_VEL
LIN {X 0,Y 350.69,Z 237.991,A -85,B 0,C 180,E1 -13740.265,E2 -13740.265} C_VEL
LIN {X 0,Y 352.845,Z 248.332,A -85,B 0,C 180,E1 -13743.017,E2 -13743.017} C_VEL
LIN {X 0,Y 353.159,Z 250.534,A -85,B 0,C 180,E1 -13743.576,E2 -13743.576} C_VEL
LIN {X 0,Y 352.153,Z 260.001,A -85,B 0,C 180,E1 -13745.761,E2 -13745.761} C_VEL
LIN {X 0,Y 357.415,Z 286.588,A -85,B 0,C 180,E1 -13746.821,E2 -13746.821} C_VEL
LIN {X 0,Y 359.343,Z 300.039,A -85,B 0,C 180,E1 -13747.275,E2 -13747.275} C_VEL
LIN {X 0,Y 357.82,Z 369.684,A -85,B 0,C 180,E1 -13748.731,E2 -13748.731} C_VEL
LIN {X 0,Y 356.921,Z 383.381,A -85,B 0,C 180,E1 -13749.241,E2 -13749.241} C_VEL
LIN {X 0,Y 355.79,Z 395.727,A -85,B 0,C 180,E1 -13749.927,E2 -13749.927} C_VEL
LIN {X 0,Y 354.358,Z 408.354,A -85,B 0,C 180,E1 -13750.898,E2 -13750.898} C_VEL
LIN {X 0,Y 352.906,Z 419.599,A -85,B 0,C 180,E1 -13752.02,E2 -13752.02} C_VEL
LIN {X 0,Y 351.493,Z 429.78,A -85,B 0,C 180,E1 -13753.296,E2 -13753.296} C_VEL
LIN {X 0,Y 350.013,Z 439.774,A -85,B 0,C 180,E1 -13754.868,E2 -13754.868} C_VEL
LIN {X 0,Y 348.781,Z 448.6,A -85,B 0,C 180,E1 -13756.6,E2 -13756.6} C_VEL
LIN {X 0,Y 347.663,Z 455.707,A -85,B 0,C 180,E1 -13758.336,E2 -13758.336} C_VEL
LIN {X 0,Y 346.998,Z 461.406,A -85,B 0,C 180,E1 -13760.086,E2 -13760.086} C_VEL
LIN {X 0,Y 346.522,Z 465.921,A -85,B 0,C 180,E1 -13761.837,E2 -13761.837} C_VEL
LIN {X 0,Y 346.206,Z 470.173,A -85,B 0,C 180,E1 -13764.103,E2 -13764.103} C_VEL
LIN {X 0,Y 346.17,Z 471.84,A -85,B 0,C 180,E1 -13765.34,E2 -13765.34} C_VEL
LIN {X 0,Y 346.163,Z 472.948,A -85,B 0,C 180,E1 -13766.506,E2 -13766.506} C_VEL
LIN {X 0,Y 346.258,Z 473.988,A -85,B 0,C 180,E1 -13768.835,E2 -13768.835} C_VEL
LIN {X 0,Y 346.32,Z 473.927,A -85,B 0,C 180,E1 -13769.998,E2 -13769.998} C_VEL
LIN {X 0,Y 346.297,Z 473.43,A -85,B 0,C 180,E1 -13771.161,E2 -13771.161} C_VEL
LIN {X 0,Y 346.188,Z 471.207,A -85,B 0,C 180,E1 -13773.489,E2 -13773.489} C_VEL
LIN {X 0,Y 346.224,Z 468.416,A -85,B 0,C 180,E1 -13775.239,E2 -13775.239} C_VEL
LIN {X 0,Y 346.338,Z 464.577,A -85,B 0,C 180,E1 -13776.991,E2 -13776.991} C_VEL
LIN {X 0,Y 346.564,Z 459.587,A -85,B 0,C 180,E1 -13778.745,E2 -13778.745} C_VEL
LIN {X 0,Y 346.977,Z 453.295,A -85,B 0,C 180,E1 -13780.5,E2 -13780.5} C_VEL
LIN {X 0,Y 347.707,Z 445.429,A -85,B 0,C 180,E1 -13782.25,E2 -13782.25} C_VEL
LIN {X 0,Y 348.483,Z 437.376,A -85,B 0,C 180,E1 -13783.704,E2 -13783.704} C_VEL
LIN {X 0,Y 349.391,Z 427.532,A -85,B 0,C 180,E1 -13785.155,E2 -13785.155} C_VEL
LIN {X 0,Y 350.341,Z 416.568,A -85,B 0,C 180,E1 -13786.457,E2 -13786.457} C_VEL
LIN {X 0,Y 351.358,Z 405.855,A -85,B 0,C 180,E1 -13787.456,E2 -13787.456} C_VEL
LIN {X 0,Y 352.371,Z 392.94,A -85,B 0,C 180,E1 -13788.38,E2 -13788.38} C_VEL
LIN {X 0,Y 353.152,Z 379.868,A -85,B 0,C 180,E1 -13789.052,E2 -13789.052} C_VEL
LIN {X 0,Y 353.696,Z 366.881,A -85,B 0,C 180,E1 -13789.474,E2 -13789.474} C_VEL
LIN {X 0,Y 354.726,Z 297.572,A -85,B 0,C 180,E1 -13790.889,E2 -13790.889} C_VEL
LIN {X 0,Y 349.814,Z 260.923,A -85,B 0,C 180,E1 -13791.927,E2 -13791.927} C_VEL
LIN {X 0,Y 351.228,Z 245.449,A -85,B 0,C 180,E1 -13795.372,E2 -13795.372} C_VEL
LIN {X 0,Y 350.543,Z 239.356,A -85,B 0,C 180,E1 -13796.809,E2 -13796.809} C_VEL
LIN {X 0,Y 347.824,Z 226.161,A -85,B 0,C 180,E1 -13800.102,E2 -13800.102} C_VEL
LIN {X 0,Y 347.729,Z 226.169,A -85,B 0,C 180,E1 -13804.46,E2 -13804.46} C_VEL
LIN {X 0,Y 347.755,Z 226.17,A -85,B 0,C 180,E1 -13807.984,E2 -13807.984} C_VEL
LIN {X 0,Y 347.729,Z 226.172,A -85,B 0,C 180,E1 -13811.826,E2 -13811.826} C_VEL
LIN {X 0,Y 347.752,Z 226.164,A -85,B 0,C 180,E1 -13815.011,E2 -13815.011} C_VEL
LIN {X 0,Y 347.76,Z 226.164,A -85,B 0,C 180,E1 -13818.387,E2 -13818.387} C_VEL
LIN {X 0,Y 347.746,Z 226.168,A -85,B 0,C 180,E1 -13822.007,E2 -13822.007} C_VEL
LIN {X 0,Y 347.713,Z 226.174,A -85,B 0,C 180,E1 -13825.532,E2 -13825.532} C_VEL
LIN {X 0,Y 347.73,Z 226.173,A -85,B 0,C 180,E1 -13829.65,E2 -13829.65} C_VEL
LIN {X 0,Y 347.816,Z 226.156,A -85,B 0,C 180,E1 -13832.742,E2 -13832.742} C_VEL
LIN {X 0,Y 347.763,Z 226.163,A -85,B 0,C 180,E1 -13836.16,E2 -13836.16} C_VEL
LIN {X 0,Y 347.796,Z 226.16,A -85,B 0,C 180,E1 -13839.908,E2 -13839.908} C_VEL
LIN {X 0,Y 347.826,Z 226.155,A -85,B 0,C 180,E1 -13842.357,E2 -13842.357} C_VEL
LIN {X 0,Y 347.857,Z 226.152,A -85,B 0,C 180,E1 -13845.969,E2 -13845.969} C_VEL
LIN {X 0,Y 347.889,Z 226.15,A -85,B 0,C 180,E1 -13849.524,E2 -13849.524} C_VEL
LIN {X 0,Y 348.032,Z 226.13,A -85,B 0,C 180,E1 -13851.873,E2 -13851.873} C_VEL
LIN {X 0,Y 348.03,Z 226.129,A -85,B 0,C 180,E1 -13854.205,E2 -13854.205} C_VEL
LIN {X 0,Y 348.16,Z 226.114,A -85,B 0,C 180,E1 -13857.686,E2 -13857.686} C_VEL
LIN {X 0,Y 348.279,Z 226.098,A -85,B 0,C 180,E1 -13860,E2 -13860} C_VEL
LIN {X 0,Y 348.157,Z 226.114,A -85,B 0,C 180,E1 -13862.313,E2 -13862.313} C_VEL
LIN {X 0,Y 348.042,Z 226.134,A -85,B 0,C 180,E1 -13866.959,E2 -13866.959} C_VEL
LIN {X 0,Y 347.885,Z 226.15,A -85,B 0,C 180,E1 -13870.475,E2 -13870.475} C_VEL
LIN {X 0,Y 347.857,Z 226.152,A -85,B 0,C 180,E1 -13874.151,E2 -13874.151} C_VEL
LIN {X 0,Y 347.803,Z 226.159,A -85,B 0,C 180,E1 -13878.268,E2 -13878.268} C_VEL
LIN {X 0,Y 347.725,Z 226.167,A -85,B 0,C 180,E1 -13881.627,E2 -13881.627} C_VEL
LIN {X 0,Y 347.771,Z 226.164,A -85,B 0,C 180,E1 -13885.111,E2 -13885.111} C_VEL
LIN {X 0,Y 347.763,Z 226.163,A -85,B 0,C 180,E1 -13887.698,E2 -13887.698} C_VEL
LIN {X 0,Y 347.705,Z 226.17,A -85,B 0,C 180,E1 -13891.703,E2 -13891.703} C_VEL
LIN {X 0,Y 347.71,Z 226.175,A -85,B 0,C 180,E1 -13894.467,E2 -13894.467} C_VEL
LIN {X 0,Y 347.739,Z 226.168,A -85,B 0,C 180,E1 -13897.991,E2 -13897.991} C_VEL
LIN {X 0,Y 347.721,Z 226.169,A -85,B 0,C 180,E1 -13901.834,E2 -13901.834} C_VEL
LIN {X 0,Y 347.677,Z 226.174,A -85,B 0,C 180,E1 -13905.031,E2 -13905.031} C_VEL
LIN {X 0,Y 347.725,Z 226.172,A -85,B 0,C 180,E1 -13908.401,E2 -13908.401} C_VEL
LIN {X 0,Y 347.751,Z 226.169,A -85,B 0,C 180,E1 -13912.015,E2 -13912.015} C_VEL
LIN {X 0,Y 347.725,Z 226.169,A -85,B 0,C 180,E1 -13915.54,E2 -13915.54} C_VEL
LIN {X 0,Y 347.728,Z 226.171,A -85,B 0,C 180,E1 -13918.304,E2 -13918.304} C_VEL
LIN {X 0,Y 347.763,Z 226.163,A -85,B 0,C 180,E1 -13920.991,E2 -13920.991} C_VEL
LIN {X 0,Y 347.817,Z 226.158,A -85,B 0,C 180,E1 -13923.611,E2 -13923.611} C_VEL
LIN {X 0,Y 347.773,Z 226.165,A -85,B 0,C 180,E1 -13926.165,E2 -13926.165} C_VEL
LIN {X 0,Y 347.79,Z 226.165,A -85,B 0,C 180,E1 -13929.912,E2 -13929.912} C_VEL
LIN {X 0,Y 347.824,Z 226.159,A -85,B 0,C 180,E1 -13933.572,E2 -13933.572} C_VEL
LIN {X 0,Y 347.884,Z 226.149,A -85,B 0,C 180,E1 -13937.164,E2 -13937.164} C_VEL
LIN {X 0,Y 347.936,Z 226.141,A -85,B 0,C 180,E1 -13940.704,E2 -13940.704} C_VEL
LIN {X 0,Y 348.029,Z 226.197,A -85,B 0,C 180,E1 -13941.786,E2 -13941.786} C_VEL
LIN {X 0,Y 348.976,Z 231.131,A -85,B 0,C 180,E1 -13943.128,E2 -13943.128} C_VEL
LIN {X 0,Y 353.379,Z 245.651,A -85,B 0,C 180,E1 -13943.674,E2 -13943.674} C_VEL
LIN {X 0,Y 355.418,Z 256.834,A -85,B 0,C 180,E1 -13944.015,E2 -13944.015} C_VEL
LIN {X 0,Y 353.885,Z 338.909,A -85,B 0,C 180,E1 -13945.696,E2 -13945.696} C_VEL
LIN {X 0,Y 353.416,Z 352.64,A -85,B 0,C 180,E1 -13946.225,E2 -13946.225} C_VEL
LIN {X 0,Y 352.793,Z 365.008,A -85,B 0,C 180,E1 -13946.933,E2 -13946.933} C_VEL
LIN {X 0,Y 352.007,Z 376.75,A -85,B 0,C 180,E1 -13947.846,E2 -13947.846} C_VEL
LIN {X 0,Y 351.012,Z 388.284,A -85,B 0,C 180,E1 -13948.998,E2 -13948.998} C_VEL
LIN {X 0,Y 350.066,Z 398.565,A -85,B 0,C 180,E1 -13950.29,E2 -13950.29} C_VEL
LIN {X 0,Y 349.145,Z 407.798,A -85,B 0,C 180,E1 -13951.732,E2 -13951.732} C_VEL
LIN {X 0,Y 348.231,Z 416.774,A -85,B 0,C 180,E1 -13953.473,E2 -13953.473} C_VEL
LIN {X 0,Y 347.53,Z 424.002,A -85,B 0,C 180,E1 -13955.223,E2 -13955.223} C_VEL
LIN {X 0,Y 347.042,Z 430.129,A -85,B 0,C 180,E1 -13957.115,E2 -13957.115} C_VEL
LIN {X 0,Y 346.663,Z 434.297,A -85,B 0,C 180,E1 -13958.747,E2 -13958.747} C_VEL
LIN {X 0,Y 346.353,Z 437.751,A -85,B 0,C 180,E1 -13960.524,E2 -13960.524} C_VEL
LIN {X 0,Y 346.264,Z 439.463,A -85,B 0,C 180,E1 -13961.711,E2 -13961.711} C_VEL
LIN {X 0,Y 346.185,Z 440.84,A -85,B 0,C 180,E1 -13962.979,E2 -13962.979} C_VEL
LIN {X 0,Y 346.081,Z 441.669,A -85,B 0,C 180,E1 -13964.105,E2 -13964.105} C_VEL
LIN {X 0,Y 346.084,Z 442.106,A -85,B 0,C 180,E1 -13965.308,E2 -13965.308} C_VEL
LIN {X 0,Y 346.21,Z 441.89,A -85,B 0,C 180,E1 -13967.43,E2 -13967.43} C_VEL
LIN {X 0,Y 346.394,Z 440.956,A -85,B 0,C 180,E1 -13968.943,E2 -13968.943} C_VEL
LIN {X 0,Y 346.87,Z 438.192,A -85,B 0,C 180,E1 -13971.25,E2 -13971.25} C_VEL
LIN {X 0,Y 347.444,Z 434.504,A -85,B 0,C 180,E1 -13973.231,E2 -13973.231} C_VEL
LIN {X 0,Y 348.191,Z 429.815,A -85,B 0,C 180,E1 -13975.079,E2 -13975.079} C_VEL
LIN {X 0,Y 349.22,Z 423.727,A -85,B 0,C 180,E1 -13976.924,E2 -13976.924} C_VEL
LIN {X 0,Y 350.429,Z 416.007,A -85,B 0,C 180,E1 -13978.772,E2 -13978.772} C_VEL
LIN {X 0,Y 351.817,Z 407.012,A -85,B 0,C 180,E1 -13980.483,E2 -13980.483} C_VEL
LIN {X 0,Y 353.2,Z 397.537,A -85,B 0,C 180,E1 -13981.92,E2 -13981.92} C_VEL
LIN {X 0,Y 353.172,Z 393.098,A -85,B 0,C 180,E1 -13982.545,E2 -13982.545} C_VEL
LIN {X 0,Y 351.471,Z 385.727,A -85,B 0,C 180,E1 -13983.586,E2 -13983.586} C_VEL
LIN {X 0,Y 349.766,Z 377.935,A -85,B 0,C 180,E1 -13984.545,E2 -13984.545} C_VEL
LIN {X 0,Y 349.686,Z 372.781,A -85,B 0,C 180,E1 -13985.031,E2 -13985.031} C_VEL
LIN {X 0,Y 350.717,Z 360.709,A -85,B 0,C 180,E1 -13985.882,E2 -13985.882} C_VEL
LIN {X 0,Y 351.598,Z 347.521,A -85,B 0,C 180,E1 -13986.532,E2 -13986.532} C_VEL
LIN {X 0,Y 352.078,Z 334.37,A -85,B 0,C 180,E1 -13986.945,E2 -13986.945} C_VEL
LIN {X 0,Y 353.911,Z 259.537,A -85,B 0,C 180,E1 -13988.493,E2 -13988.493} C_VEL
LIN {X 0,Y 349.437,Z 248.256,A -85,B 0,C 180,E1 -13989.146,E2 -13989.146} C_VEL
LIN {X 0,Y 342.692,Z 233.881,A -85,B 0,C 180,E1 -13990.109,E2 -13990.109} C_VEL
LIN {X 0,Y 342.041,Z 232.165,A -85,B 0,C 180,E1 -13990.248,E2 -13990.248} C_VEL
LIN {X 0,Y 340.737,Z 227.037,A -85,B 0,C 180,E1 -13991.882,E2 -13991.882} C_VEL
LIN {X 0,Y 340.772,Z 227.037,A -85,B 0,C 180,E1 -13995.476,E2 -13995.476} C_VEL
LIN {X 0,Y 340.715,Z 227.045,A -85,B 0,C 180,E1 -13998.695,E2 -13998.695} C_VEL
LIN {X 0,Y 340.723,Z 227.042,A -85,B 0,C 180,E1 -14001.772,E2 -14001.772} C_VEL
LIN {X 0,Y 340.709,Z 227.039,A -85,B 0,C 180,E1 -14005.595,E2 -14005.595} C_VEL
LIN {X 0,Y 340.689,Z 227.042,A -85,B 0,C 180,E1 -14008.955,E2 -14008.955} C_VEL
LIN {X 0,Y 340.763,Z 227.035,A -85,B 0,C 180,E1 -14012.474,E2 -14012.474} C_VEL
LIN {X 0,Y 340.742,Z 227.032,A -85,B 0,C 180,E1 -14015.638,E2 -14015.638} C_VEL
LIN {X 0,Y 340.748,Z 227.031,A -85,B 0,C 180,E1 -14019.475,E2 -14019.475} C_VEL
LIN {X 0,Y 340.84,Z 227.023,A -85,B 0,C 180,E1 -14021.984,E2 -14021.984} C_VEL
LIN {X 0,Y 340.834,Z 227.029,A -85,B 0,C 180,E1 -14025.716,E2 -14025.716} C_VEL
LIN {X 0,Y 340.848,Z 227.027,A -85,B 0,C 180,E1 -14029.306,E2 -14029.306} C_VEL
LIN {X 0,Y 341.039,Z 226.995,A -85,B 0,C 180,E1 -14032.898,E2 -14032.898} C_VEL
LIN {X 0,Y 341.142,Z 226.985,A -85,B 0,C 180,E1 -14037.639,E2 -14037.639} C_VEL
LIN {X 0,Y 341.234,Z 226.97,A -85,B 0,C 180,E1 -14040,E2 -14040} C_VEL
LIN {X 0,Y 341.142,Z 226.981,A -85,B 0,C 180,E1 -14042.362,E2 -14042.362} C_VEL
LIN {X 0,Y 340.997,Z 227.001,A -85,B 0,C 180,E1 -14047.104,E2 -14047.104} C_VEL
LIN {X 0,Y 340.83,Z 227.017,A -85,B 0,C 180,E1 -14050.695,E2 -14050.695} C_VEL
LIN {X 0,Y 340.846,Z 227.019,A -85,B 0,C 180,E1 -14054.326,E2 -14054.326} C_VEL
LIN {X 0,Y 340.752,Z 227.034,A -85,B 0,C 180,E1 -14058.433,E2 -14058.433} C_VEL
LIN {X 0,Y 340.703,Z 227.043,A -85,B 0,C 180,E1 -14061.843,E2 -14061.843} C_VEL
LIN {X 0,Y 340.704,Z 227.044,A -85,B 0,C 180,E1 -14065.67,E2 -14065.67} C_VEL
LIN {X 0,Y 340.688,Z 227.046,A -85,B 0,C 180,E1 -14069.676,E2 -14069.676} C_VEL
LIN {X 0,Y 340.666,Z 227.05,A -85,B 0,C 180,E1 -14072.438,E2 -14072.438} C_VEL
LIN {X 0,Y 340.703,Z 227.044,A -85,B 0,C 180,E1 -14075.281,E2 -14075.281} C_VEL
LIN {X 0,Y 340.683,Z 227.046,A -85,B 0,C 180,E1 -14078.384,E2 -14078.384} C_VEL
LIN {X 0,Y 340.688,Z 227.031,A -85,B 0,C 180,E1 -14082.046,E2 -14082.046} C_VEL
LIN {X 0,Y 340.645,Z 227.054,A -85,B 0,C 180,E1 -14086.229,E2 -14086.229} C_VEL
LIN {X 0,Y 340.666,Z 227.05,A -85,B 0,C 180,E1 -14088.689,E2 -14088.689} C_VEL
LIN {X 0,Y 340.715,Z 227.047,A -85,B 0,C 180,E1 -14091.772,E2 -14091.772} C_VEL
LIN {X 0,Y 340.721,Z 227.04,A -85,B 0,C 180,E1 -14095.597,E2 -14095.597} C_VEL
LIN {X 0,Y 340.735,Z 227.173,A -85,B 0,C 180,E1 -14096.382,E2 -14096.382} C_VEL
LIN {X 0,Y 343.472,Z 238.123,A -85,B 0,C 180,E1 -14099.583,E2 -14099.583} C_VEL
LIN {X 0,Y 345.713,Z 248.579,A -85,B 0,C 180,E1 -14102.453,E2 -14102.453} C_VEL
LIN {X 0,Y 346.316,Z 252.52,A -85,B 0,C 180,E1 -14103.484,E2 -14103.484} C_VEL
LIN {X 0,Y 345.486,Z 259.708,A -85,B 0,C 180,E1 -14105.176,E2 -14105.176} C_VEL
LIN {X 0,Y 351.098,Z 287.622,A -85,B 0,C 180,E1 -14106.32,E2 -14106.32} C_VEL
LIN {X 0,Y 353.006,Z 300.997,A -85,B 0,C 180,E1 -14106.784,E2 -14106.784} C_VEL
LIN {X 0,Y 351.442,Z 368.553,A -85,B 0,C 180,E1 -14108.21,E2 -14108.21} C_VEL
LIN {X 0,Y 350.58,Z 381.758,A -85,B 0,C 180,E1 -14108.694,E2 -14108.694} C_VEL
LIN {X 0,Y 349.39,Z 394.448,A -85,B 0,C 180,E1 -14109.389,E2 -14109.389} C_VEL
LIN {X 0,Y 348.067,Z 405.764,A -85,B 0,C 180,E1 -14110.232,E2 -14110.232} C_VEL
LIN {X 0,Y 346.532,Z 417.431,A -85,B 0,C 180,E1 -14111.371,E2 -14111.371} C_VEL
LIN {X 0,Y 344.988,Z 427.932,A -85,B 0,C 180,E1 -14112.666,E2 -14112.666} C_VEL
LIN {X 0,Y 343.567,Z 437.363,A -85,B 0,C 180,E1 -14114.11,E2 -14114.11} C_VEL
LIN {X 0,Y 342.322,Z 445.921,A -85,B 0,C 180,E1 -14115.737,E2 -14115.737} C_VEL
LIN {X 0,Y 341.046,Z 453.449,A -85,B 0,C 180,E1 -14117.503,E2 -14117.503} C_VEL
LIN {X 0,Y 340.203,Z 459.534,A -85,B 0,C 180,E1 -14119.284,E2 -14119.284} C_VEL
LIN {X 0,Y 339.61,Z 464.38,A -85,B 0,C 180,E1 -14121.07,E2 -14121.07} C_VEL
LIN {X 0,Y 339.253,Z 468.124,A -85,B 0,C 180,E1 -14122.858,E2 -14122.858} C_VEL
LIN {X 0,Y 339.131,Z 470.176,A -85,B 0,C 180,E1 -14124.12,E2 -14124.12} C_VEL
LIN {X 0,Y 339.072,Z 471.592,A -85,B 0,C 180,E1 -14125.243,E2 -14125.243} C_VEL
LIN {X 0,Y 339.086,Z 472.672,A -85,B 0,C 180,E1 -14126.433,E2 -14126.433} C_VEL
LIN {X 0,Y 339.16,Z 473.67,A -85,B 0,C 180,E1 -14128.811,E2 -14128.811} C_VEL
LIN {X 0,Y 339.227,Z 473.58,A -85,B 0,C 180,E1 -14129.998,E2 -14129.998} C_VEL
LIN {X 0,Y 339.201,Z 473.048,A -85,B 0,C 180,E1 -14131.185,E2 -14131.185} C_VEL
LIN {X 0,Y 339.114,Z 470.784,A -85,B 0,C 180,E1 -14133.562,E2 -14133.562} C_VEL
LIN {X 0,Y 339.135,Z 467.68,A -85,B 0,C 180,E1 -14135.495,E2 -14135.495} C_VEL
LIN {X 0,Y 339.261,Z 464.058,A -85,B 0,C 180,E1 -14137.137,E2 -14137.137} C_VEL
LIN {X 0,Y 339.51,Z 459.015,A -85,B 0,C 180,E1 -14138.929,E2 -14138.929} C_VEL
LIN {X 0,Y 339.928,Z 452.662,A -85,B 0,C 180,E1 -14140.721,E2 -14140.721} C_VEL
LIN {X 0,Y 340.732,Z 444.701,A -85,B 0,C 180,E1 -14142.505,E2 -14142.505} C_VEL
LIN {X 0,Y 341.563,Z 436.569,A -85,B 0,C 180,E1 -14143.987,E2 -14143.987} C_VEL
LIN {X 0,Y 342.478,Z 426.625,A -85,B 0,C 180,E1 -14145.469,E2 -14145.469} C_VEL
LIN {X 0,Y 343.483,Z 415.483,A -85,B 0,C 180,E1 -14146.795,E2 -14146.795} C_VEL
LIN {X 0,Y 344.494,Z 404.563,A -85,B 0,C 180,E1 -14147.815,E2 -14147.815} C_VEL
LIN {X 0,Y 345.495,Z 392.527,A -85,B 0,C 180,E1 -14148.682,E2 -14148.682} C_VEL
LIN {X 0,Y 346.316,Z 379.408,A -85,B 0,C 180,E1 -14149.366,E2 -14149.366} C_VEL
LIN {X 0,Y 346.878,Z 366.336,A -85,B 0,C 180,E1 -14149.796,E2 -14149.796} C_VEL
LIN {X 0,Y 347.881,Z 297.969,A -85,B 0,C 180,E1 -14151.221,E2 -14151.221} C_VEL
LIN {X 0,Y 342.884,Z 260.562,A -85,B 0,C 180,E1 -14152.312,E2 -14152.312} C_VEL
LIN {X 0,Y 344.217,Z 247.023,A -85,B 0,C 180,E1 -14155.384,E2 -14155.384} C_VEL
LIN {X 0,Y 343.997,Z 243.186,A -85,B 0,C 180,E1 -14156.294,E2 -14156.294} C_VEL
LIN {X 0,Y 341.974,Z 232.831,A -85,B 0,C 180,E1 -14158.873,E2 -14158.873} C_VEL
LIN {X 0,Y 340.749,Z 227.04,A -85,B 0,C 180,E1 -14160.391,E2 -14160.391} C_VEL
LIN {X 0,Y 340.707,Z 227.044,A -85,B 0,C 180,E1 -14164.4,E2 -14164.4} C_VEL
LIN {X 0,Y 340.691,Z 227.046,A -85,B 0,C 180,E1 -14168.381,E2 -14168.381} C_VEL
LIN {X 0,Y 340.678,Z 227.05,A -85,B 0,C 180,E1 -14172.041,E2 -14172.041} C_VEL
LIN {X 0,Y 340.688,Z 227.046,A -85,B 0,C 180,E1 -14176.212,E2 -14176.212} C_VEL
LIN {X 0,Y 340.738,Z 227.044,A -85,B 0,C 180,E1 -14179.734,E2 -14179.734} C_VEL
LIN {X 0,Y 340.68,Z 227.05,A -85,B 0,C 180,E1 -14183.555,E2 -14183.555} C_VEL
LIN {X 0,Y 340.661,Z 227.049,A -85,B 0,C 180,E1 -14186.149,E2 -14186.149} C_VEL
LIN {X 0,Y 340.74,Z 227.038,A -85,B 0,C 180,E1 -14190.329,E2 -14190.329} C_VEL
LIN {X 0,Y 340.769,Z 227.035,A -85,B 0,C 180,E1 -14193.017,E2 -14193.017} C_VEL
LIN {X 0,Y 340.704,Z 227.043,A -85,B 0,C 180,E1 -14196.925,E2 -14196.925} C_VEL
LIN {X 0,Y 340.763,Z 227.035,A -85,B 0,C 180,E1 -14200.732,E2 -14200.732} C_VEL
LIN {X 0,Y 340.746,Z 227.041,A -85,B 0,C 180,E1 -14203.216,E2 -14203.216} C_VEL
LIN {X 0,Y 340.804,Z 227.032,A -85,B 0,C 180,E1 -14206.889,E2 -14206.889} C_VEL
LIN {X 0,Y 340.887,Z 227.02,A -85,B 0,C 180,E1 -14210.506,E2 -14210.506} C_VEL
LIN {X 0,Y 341.04,Z 227.003,A -85,B 0,C 180,E1 -14212.897,E2 -14212.897} C_VEL
LIN {X 0,Y 341.122,Z 226.991,A -85,B 0,C 180,E1 -14217.638,E2 -14217.638} C_VEL
LIN {X 0,Y 341.23,Z 226.976,A -85,B 0,C 180,E1 -14220,E2 -14220} C_VEL
LIN {X 0,Y 341.119,Z 226.991,A -85,B 0,C 180,E1 -14222.361,E2 -14222.361} C_VEL
LIN {X 0,Y 341.011,Z 227.008,A -85,B 0,C 180,E1 -14227.103,E2 -14227.103} C_VEL
LIN {X 0,Y 340.828,Z 227.031,A -85,B 0,C 180,E1 -14230.695,E2 -14230.695} C_VEL
LIN {X 0,Y 340.822,Z 227.029,A -85,B 0,C 180,E1 -14234.326,E2 -14234.326} C_VEL
LIN {X 0,Y 340.756,Z 227.038,A -85,B 0,C 180,E1 -14238.447,E2 -14238.447} C_VEL
LIN {X 0,Y 340.679,Z 227.045,A -85,B 0,C 180,E1 -14241.844,E2 -14241.844} C_VEL
LIN {X 0,Y 340.732,Z 227.038,A -85,B 0,C 180,E1 -14245.667,E2 -14245.667} C_VEL
LIN {X 0,Y 340.681,Z 227.048,A -85,B 0,C 180,E1 -14248.325,E2 -14248.325} C_VEL
LIN {X 0,Y 340.655,Z 227.049,A -85,B 0,C 180,E1 -14251.049,E2 -14251.049} C_VEL
LIN {X 0,Y 340.684,Z 227.045,A -85,B 0,C 180,E1 -14255.282,E2 -14255.282} C_VEL
LIN {X 0,Y 340.677,Z 227.051,A -85,B 0,C 180,E1 -14258.389,E2 -14258.389} C_VEL
LIN {X 0,Y 340.669,Z 227.049,A -85,B 0,C 180,E1 -14262.049,E2 -14262.049} C_VEL
LIN {X 0,Y 340.626,Z 227.057,A -85,B 0,C 180,E1 -14266.231,E2 -14266.231} C_VEL
LIN {X 0,Y 340.664,Z 227.049,A -85,B 0,C 180,E1 -14269.757,E2 -14269.757} C_VEL
LIN {X 0,Y 340.684,Z 227.044,A -85,B 0,C 180,E1 -14273.262,E2 -14273.262} C_VEL
LIN {X 0,Y 340.674,Z 227.052,A -85,B 0,C 180,E1 -14276.157,E2 -14276.157} C_VEL
LIN {X 0,Y 340.726,Z 227.043,A -85,B 0,C 180,E1 -14280.333,E2 -14280.333} C_VEL
LIN {X 0,Y 340.789,Z 227.032,A -85,B 0,C 180,E1 -14283.024,E2 -14283.024} C_VEL
LIN {X 0,Y 340.742,Z 227.04,A -85,B 0,C 180,E1 -14285.642,E2 -14285.642} C_VEL
LIN {X 0,Y 340.72,Z 227.042,A -85,B 0,C 180,E1 -14289.477,E2 -14289.477} C_VEL
LIN {X 0,Y 340.784,Z 227.037,A -85,B 0,C 180,E1 -14291.984,E2 -14291.984} C_VEL
LIN {X 0,Y 340.863,Z 227.028,A -85,B 0,C 180,E1 -14295.708,E2 -14295.708} C_VEL
LIN {X 0,Y 340.865,Z 227.024,A -85,B 0,C 180,E1 -14299.309,E2 -14299.309} C_VEL
LIN {X 0,Y 340.972,Z 227.028,A -85,B 0,C 180,E1 -14301.512,E2 -14301.512} C_VEL
LIN {X 0,Y 341.841,Z 231.405,A -85,B 0,C 180,E1 -14302.727,E2 -14302.727} C_VEL
LIN {X 0,Y 346.802,Z 247.501,A -85,B 0,C 180,E1 -14303.365,E2 -14303.365} C_VEL
LIN {X 0,Y 348.655,Z 257.523,A -85,B 0,C 180,E1 -14303.679,E2 -14303.679} C_VEL
LIN {X 0,Y 347.055,Z 339.551,A -85,B 0,C 180,E1 -14305.393,E2 -14305.393} C_VEL
LIN {X 0,Y 346.572,Z 353.179,A -85,B 0,C 180,E1 -14305.932,E2 -14305.932} C_VEL
LIN {X 0,Y 345.925,Z 365.487,A -85,B 0,C 180,E1 -14306.654,E2 -14306.654} C_VEL
LIN {X 0,Y 345.046,Z 378.098,A -85,B 0,C 180,E1 -14307.668,E2 -14307.668} C_VEL
LIN {X 0,Y 344.052,Z 389.342,A -85,B 0,C 180,E1 -14308.832,E2 -14308.832} C_VEL
LIN {X 0,Y 343.064,Z 399.464,A -85,B 0,C 180,E1 -14310.149,E2 -14310.149} C_VEL
LIN {X 0,Y 342.017,Z 409.41,A -85,B 0,C 180,E1 -14311.768,E2 -14311.768} C_VEL
LIN {X 0,Y 341.127,Z 418.16,A -85,B 0,C 180,E1 -14313.545,E2 -14313.545} C_VEL
LIN {X 0,Y 340.392,Z 425.145,A -85,B 0,C 180,E1 -14315.333,E2 -14315.333} C_VEL
LIN {X 0,Y 339.968,Z 430.721,A -85,B 0,C 180,E1 -14317.126,E2 -14317.126} C_VEL
LIN {X 0,Y 339.534,Z 435.122,A -85,B 0,C 180,E1 -14318.932,E2 -14318.932} C_VEL
LIN {X 0,Y 339.234,Z 438.439,A -85,B 0,C 180,E1 -14320.747,E2 -14320.747} C_VEL
LIN {X 0,Y 339.091,Z 441.217,A -85,B 0,C 180,E1 -14323.065,E2 -14323.065} C_VEL
LIN {X 0,Y 338.979,Z 442.103,A -85,B 0,C 180,E1 -14324.407,E2 -14324.407} C_VEL
LIN {X 0,Y 338.992,Z 442.473,A -85,B 0,C 180,E1 -14325.636,E2 -14325.636} C_VEL
LIN {X 0,Y 339.142,Z 442.208,A -85,B 0,C 180,E1 -14327.59,E2 -14327.59} C_VEL
LIN {X 0,Y 339.376,Z 441.06,A -85,B 0,C 180,E1 -14329.35,E2 -14329.35} C_VEL
LIN {X 0,Y 339.834,Z 438.51,A -85,B 0,C 180,E1 -14331.468,E2 -14331.468} C_VEL
LIN {X 0,Y 340.561,Z 434.286,A -85,B 0,C 180,E1 -14333.729,E2 -14333.729} C_VEL
LIN {X 0,Y 341.406,Z 429.412,A -85,B 0,C 180,E1 -14335.613,E2 -14335.613} C_VEL
LIN {X 0,Y 342.473,Z 423.142,A -85,B 0,C 180,E1 -14337.498,E2 -14337.498} C_VEL
LIN {X 0,Y 343.847,Z 415.233,A -85,B 0,C 180,E1 -14339.376,E2 -14339.376} C_VEL
LIN {X 0,Y 345.371,Z 405.67,A -85,B 0,C 180,E1 -14341.155,E2 -14341.155} C_VEL
LIN {X 0,Y 346.848,Z 395.645,A -85,B 0,C 180,E1 -14342.648,E2 -14342.648} C_VEL
LIN {X 0,Y 348.342,Z 385.251,A -85,B 0,C 180,E1 -14343.872,E2 -14343.872} C_VEL
LIN {X 0,Y 349.594,Z 373.702,A -85,B 0,C 180,E1 -14344.955,E2 -14344.955} C_VEL
LIN {X 0,Y 349.686,Z 372.781,A -85,B 0,C 180,E1 -14345.031,E2 -14345.031} C_VEL
LIN {X 0,Y 349.592,Z 367.549,A -85,B 0,C 180,E1 -14345.485,E2 -14345.485} C_VEL
LIN {X 0,Y 347.727,Z 358.988,A -85,B 0,C 180,E1 -14346.254,E2 -14346.254} C_VEL
LIN {X 0,Y 345.713,Z 350.15,A -85,B 0,C 180,E1 -14346.908,E2 -14346.908} C_VEL
LIN {X 0,Y 345.364,Z 344.494,A -85,B 0,C 180,E1 -14347.175,E2 -14347.175} C_VEL
LIN {X 0,Y 345.821,Z 328.821,A -85,B 0,C 180,E1 -14347.591,E2 -14347.591} C_VEL
LIN {X 0,Y 347.597,Z 260.796,A -85,B 0,C 180,E1 -14349.019,E2 -14349.019} C_VEL
LIN {X 0,Y 339.793,Z 242.769,A -85,B 0,C 180,E1 -14350.175,E2 -14350.175} C_VEL
LIN {X 0,Y 334.896,Z 232.595,A -85,B 0,C 180,E1 -14350.933,E2 -14350.933} C_VEL
LIN {X 0,Y 333.697,Z 227.919,A -85,B 0,C 180,E1 -14352.513,E2 -14352.513} C_VEL
LIN {X 0,Y 333.719,Z 227.916,A -85,B 0,C 180,E1 -14355.976,E2 -14355.976} C_VEL
LIN {X 0,Y 333.692,Z 227.919,A -85,B 0,C 180,E1 -14359.304,E2 -14359.304} C_VEL
LIN {X 0,Y 333.653,Z 227.922,A -85,B 0,C 180,E1 -14363.167,E2 -14363.167} C_VEL
LIN {X 0,Y 333.623,Z 227.926,A -85,B 0,C 180,E1 -14366.791,E2 -14366.791} C_VEL
LIN {X 0,Y 333.689,Z 227.918,A -85,B 0,C 180,E1 -14369.71,E2 -14369.71} C_VEL
LIN {X 0,Y 333.727,Z 227.91,A -85,B 0,C 180,E1 -14372.4,E2 -14372.4} C_VEL
LIN {X 0,Y 333.711,Z 227.906,A -85,B 0,C 180,E1 -14375.09,E2 -14375.09} C_VEL
LIN {X 0,Y 333.677,Z 227.91,A -85,B 0,C 180,E1 -14379.019,E2 -14379.019} C_VEL
LIN {X 0,Y 333.777,Z 227.907,A -85,B 0,C 180,E1 -14381.589,E2 -14381.589} C_VEL
LIN {X 0,Y 333.791,Z 227.908,A -85,B 0,C 180,E1 -14385.577,E2 -14385.577} C_VEL
LIN {X 0,Y 333.812,Z 227.901,A -85,B 0,C 180,E1 -14389.078,E2 -14389.078} C_VEL
LIN {X 0,Y 333.987,Z 227.873,A -85,B 0,C 180,E1 -14392.747,E2 -14392.747} C_VEL
LIN {X 0,Y 333.784,Z 227.903,A -85,B 0,C 180,E1 -14395.169,E2 -14395.169} C_VEL
LIN {X 0,Y 334.08,Z 227.863,A -85,B 0,C 180,E1 -14397.589,E2 -14397.589} C_VEL
LIN {X 0,Y 334.186,Z 227.848,A -85,B 0,C 180,E1 -14400,E2 -14400} C_VEL
LIN {X 0,Y 334.079,Z 227.861,A -85,B 0,C 180,E1 -14402.412,E2 -14402.412} C_VEL
LIN {X 0,Y 333.977,Z 227.869,A -85,B 0,C 180,E1 -14406.04,E2 -14406.04} C_VEL
LIN {X 0,Y 333.801,Z 227.892,A -85,B 0,C 180,E1 -14409.697,E2 -14409.697} C_VEL
LIN {X 0,Y 333.775,Z 227.901,A -85,B 0,C 180,E1 -14413.393,E2 -14413.393} C_VEL
LIN {X 0,Y 333.738,Z 227.906,A -85,B 0,C 180,E1 -14415.889,E2 -14415.889} C_VEL
LIN {X 0,Y 333.641,Z 227.918,A -85,B 0,C 180,E1 -14419.697,E2 -14419.697} C_VEL
LIN {X 0,Y 333.641,Z 227.918,A -85,B 0,C 180,E1 -14423.593,E2 -14423.593} C_VEL
LIN {X 0,Y 333.641,Z 227.925,A -85,B 0,C 180,E1 -14426.255,E2 -14426.255} C_VEL
LIN {X 0,Y 333.646,Z 227.923,A -85,B 0,C 180,E1 -14430.278,E2 -14430.278} C_VEL
LIN {X 0,Y 333.621,Z 227.926,A -85,B 0,C 180,E1 -14433.211,E2 -14433.211} C_VEL
LIN {X 0,Y 333.662,Z 227.923,A -85,B 0,C 180,E1 -14436.141,E2 -14436.141} C_VEL
LIN {X 0,Y 333.623,Z 227.927,A -85,B 0,C 180,E1 -14439.196,E2 -14439.196} C_VEL
LIN {X 0,Y 333.622,Z 227.913,A -85,B 0,C 180,E1 -14442.501,E2 -14442.501} C_VEL
LIN {X 0,Y 333.589,Z 227.931,A -85,B 0,C 180,E1 -14445.956,E2 -14445.956} C_VEL
LIN {X 0,Y 333.598,Z 227.926,A -85,B 0,C 180,E1 -14449.326,E2 -14449.326} C_VEL
LIN {X 0,Y 333.659,Z 227.916,A -85,B 0,C 180,E1 -14453.17,E2 -14453.17} C_VEL
LIN {X 0,Y 333.7,Z 228.119,A -85,B 0,C 180,E1 -14455.803,E2 -14455.803} C_VEL
LIN {X 0,Y 336.564,Z 239.499,A -85,B 0,C 180,E1 -14459.225,E2 -14459.225} C_VEL
LIN {X 0,Y 338.827,Z 249.98,A -85,B 0,C 180,E1 -14462.18,E2 -14462.18} C_VEL
LIN {X 0,Y 339.452,Z 253.687,A -85,B 0,C 180,E1 -14463.178,E2 -14463.178} C_VEL
LIN {X 0,Y 338.865,Z 259.331,A -85,B 0,C 180,E1 -14464.545,E2 -14464.545} C_VEL
LIN {X 0,Y 344.483,Z 286.995,A -85,B 0,C 180,E1 -14465.728,E2 -14465.728} C_VEL
LIN {X 0,Y 346.663,Z 301.485,A -85,B 0,C 180,E1 -14466.259,E2 -14466.259} C_VEL
LIN {X 0,Y 345.052,Z 368.548,A -85,B 0,C 180,E1 -14467.706,E2 -14467.706} C_VEL
LIN {X 0,Y 344.136,Z 381.645,A -85,B 0,C 180,E1 -14468.196,E2 -14468.196} C_VEL
LIN {X 0,Y 342.931,Z 394.275,A -85,B 0,C 180,E1 -14468.904,E2 -14468.904} C_VEL
LIN {X 0,Y 341.432,Z 406.345,A -85,B 0,C 180,E1 -14469.831,E2 -14469.831} C_VEL
LIN {X 0,Y 339.842,Z 417.834,A -85,B 0,C 180,E1 -14470.991,E2 -14470.991} C_VEL
LIN {X 0,Y 338.229,Z 428.21,A -85,B 0,C 180,E1 -14472.308,E2 -14472.308} C_VEL
LIN {X 0,Y 336.669,Z 437.933,A -85,B 0,C 180,E1 -14473.854,E2 -14473.854} C_VEL
LIN {X 0,Y 335.423,Z 445.976,A -85,B 0,C 180,E1 -14475.437,E2 -14475.437} C_VEL
LIN {X 0,Y 334.114,Z 453.437,A -85,B 0,C 180,E1 -14477.239,E2 -14477.239} C_VEL
LIN {X 0,Y 333.201,Z 459.457,A -85,B 0,C 180,E1 -14479.056,E2 -14479.056} C_VEL
LIN {X 0,Y 332.572,Z 464.245,A -85,B 0,C 180,E1 -14480.879,E2 -14480.879} C_VEL
LIN {X 0,Y 332.18,Z 467.937,A -85,B 0,C 180,E1 -14482.706,E2 -14482.706} C_VEL
LIN {X 0,Y 332.03,Z 470.201,A -85,B 0,C 180,E1 -14484.18,E2 -14484.18} C_VEL
LIN {X 0,Y 332.009,Z 472.397,A -85,B 0,C 180,E1 -14486.357,E2 -14486.357} C_VEL
LIN {X 0,Y 332.062,Z 473.352,A -85,B 0,C 180,E1 -14488.785,E2 -14488.785} C_VEL
LIN {X 0,Y 332.136,Z 473.224,A -85,B 0,C 180,E1 -14489.998,E2 -14489.998} C_VEL
LIN {X 0,Y 332.104,Z 472.667,A -85,B 0,C 180,E1 -14491.21,E2 -14491.21} C_VEL
LIN {X 0,Y 332.04,Z 470.36,A -85,B 0,C 180,E1 -14493.638,E2 -14493.638} C_VEL
LIN {X 0,Y 332.082,Z 468.555,A -85,B 0,C 180,E1 -14494.854,E2 -14494.854} C_VEL
LIN {X 0,Y 332.156,Z 464.984,A -85,B 0,C 180,E1 -14496.68,E2 -14496.68} C_VEL
LIN {X 0,Y 332.344,Z 460.279,A -85,B 0,C 180,E1 -14498.51,E2 -14498.51} C_VEL
LIN {X 0,Y 332.77,Z 454.305,A -85,B 0,C 180,E1 -14500.339,E2 -14500.339} C_VEL
LIN {X 0,Y 333.455,Z 446.844,A -85,B 0,C 180,E1 -14502.164,E2 -14502.164} C_VEL
LIN {X 0,Y 334.417,Z 437.558,A -85,B 0,C 180,E1 -14503.982,E2 -14503.982} C_VEL
LIN {X 0,Y 335.403,Z 427.38,A -85,B 0,C 180,E1 -14505.563,E2 -14505.563} C_VEL
LIN {X 0,Y 336.369,Z 417.116,A -85,B 0,C 180,E1 -14506.848,E2 -14506.848} C_VEL
LIN {X 0,Y 337.436,Z 406.744,A -85,B 0,C 180,E1 -14507.887,E2 -14507.887} C_VEL
LIN {X 0,Y 338.475,Z 394.342,A -85,B 0,C 180,E1 -14508.849,E2 -14508.849} C_VEL
LIN {X 0,Y 339.368,Z 381.284,A -85,B 0,C 180,E1 -14509.582,E2 -14509.582} C_VEL
LIN {X 0,Y 340.002,Z 368.587,A -85,B 0,C 180,E1 -14510.056,E2 -14510.056} C_VEL
LIN {X 0,Y 341.12,Z 298.843,A -85,B 0,C 180,E1 -14511.545,E2 -14511.545} C_VEL
LIN {X 0,Y 335.992,Z 260.32,A -85,B 0,C 180,E1 -14512.68,E2 -14512.68} C_VEL
LIN {X 0,Y 337.255,Z 247.657,A -85,B 0,C 180,E1 -14515.616,E2 -14515.616} C_VEL
LIN {X 0,Y 336.606,Z 241.832,A -85,B 0,C 180,E1 -14517.047,E2 -14517.047} C_VEL
LIN {X 0,Y 333.707,Z 227.916,A -85,B 0,C 180,E1 -14520.657,E2 -14520.657} C_VEL
LIN {X 0,Y 333.67,Z 227.919,A -85,B 0,C 180,E1 -14524.769,E2 -14524.769} C_VEL
LIN {X 0,Y 333.634,Z 227.926,A -85,B 0,C 180,E1 -14527.647,E2 -14527.647} C_VEL
LIN {X 0,Y 333.627,Z 227.924,A -85,B 0,C 180,E1 -14530.763,E2 -14530.763} C_VEL
LIN {X 0,Y 333.608,Z 227.928,A -85,B 0,C 180,E1 -14534.252,E2 -14534.252} C_VEL
LIN {X 0,Y 333.67,Z 227.923,A -85,B 0,C 180,E1 -14537.622,E2 -14537.622} C_VEL
LIN {X 0,Y 333.652,Z 227.922,A -85,B 0,C 180,E1 -14541.192,E2 -14541.192} C_VEL
LIN {X 0,Y 333.654,Z 227.922,A -85,B 0,C 180,E1 -14545.222,E2 -14545.222} C_VEL
LIN {X 0,Y 333.665,Z 227.924,A -85,B 0,C 180,E1 -14549.634,E2 -14549.634} C_VEL
LIN {X 0,Y 333.708,Z 227.914,A -85,B 0,C 180,E1 -14552.398,E2 -14552.398} C_VEL
LIN {X 0,Y 333.696,Z 227.917,A -85,B 0,C 180,E1 -14555.088,E2 -14555.088} C_VEL
LIN {X 0,Y 333.679,Z 227.919,A -85,B 0,C 180,E1 -14559.019,E2 -14559.019} C_VEL
LIN {X 0,Y 333.755,Z 227.911,A -85,B 0,C 180,E1 -14561.587,E2 -14561.587} C_VEL
LIN {X 0,Y 333.768,Z 227.909,A -85,B 0,C 180,E1 -14565.575,E2 -14565.575} C_VEL
LIN {X 0,Y 333.794,Z 227.906,A -85,B 0,C 180,E1 -14569.076,E2 -14569.076} C_VEL
LIN {X 0,Y 333.989,Z 227.88,A -85,B 0,C 180,E1 -14572.746,E2 -14572.746} C_VEL
LIN {X 0,Y 333.769,Z 227.911,A -85,B 0,C 180,E1 -14575.168,E2 -14575.168} C_VEL
LIN {X 0,Y 334.06,Z 227.869,A -85,B 0,C 180,E1 -14577.588,E2 -14577.588} C_VEL
LIN {X 0,Y 334.181,Z 227.852,A -85,B 0,C 180,E1 -14580,E2 -14580} C_VEL
LIN {X 0,Y 334.057,Z 227.869,A -85,B 0,C 180,E1 -14582.411,E2 -14582.411} C_VEL
LIN {X 0,Y 333.944,Z 227.884,A -85,B 0,C 180,E1 -14586.721,E2 -14586.721} C_VEL
LIN {X 0,Y 333.807,Z 227.901,A -85,B 0,C 180,E1 -14589.696,E2 -14589.696} C_VEL
LIN {X 0,Y 333.751,Z 227.909,A -85,B 0,C 180,E1 -14593.393,E2 -14593.393} C_VEL
LIN {X 0,Y 333.687,Z 227.918,A -85,B 0,C 180,E1 -14597.149,E2 -14597.149} C_VEL
LIN {X 0,Y 333.622,Z 227.924,A -85,B 0,C 180,E1 -14599.697,E2 -14599.697} C_VEL
LIN {X 0,Y 333.629,Z 227.924,A -85,B 0,C 180,E1 -14603.593,E2 -14603.593} C_VEL
LIN {X 0,Y 333.691,Z 227.918,A -85,B 0,C 180,E1 -14606.25,E2 -14606.25} C_VEL
LIN {X 0,Y 333.634,Z 227.923,A -85,B 0,C 180,E1 -14608.979,E2 -14608.979} C_VEL
LIN {X 0,Y 333.602,Z 227.926,A -85,B 0,C 180,E1 -14613.212,E2 -14613.212} C_VEL
LIN {X 0,Y 333.643,Z 227.924,A -85,B 0,C 180,E1 -14616.143,E2 -14616.143} C_VEL
LIN {X 0,Y 333.616,Z 227.925,A -85,B 0,C 180,E1 -14619.196,E2 -14619.196} C_VEL
LIN {X 0,Y 333.604,Z 227.929,A -85,B 0,C 180,E1 -14622.503,E2 -14622.503} C_VEL
LIN {X 0,Y 333.569,Z 227.933,A -85,B 0,C 180,E1 -14625.959,E2 -14625.959} C_VEL
LIN {X 0,Y 333.624,Z 227.924,A -85,B 0,C 180,E1 -14629.32,E2 -14629.32} C_VEL
LIN {X 0,Y 333.644,Z 227.921,A -85,B 0,C 180,E1 -14633.172,E2 -14633.172} C_VEL
LIN {X 0,Y 333.619,Z 227.925,A -85,B 0,C 180,E1 -14636.796,E2 -14636.796} C_VEL
LIN {X 0,Y 333.679,Z 227.919,A -85,B 0,C 180,E1 -14639.717,E2 -14639.717} C_VEL
LIN {X 0,Y 333.725,Z 227.914,A -85,B 0,C 180,E1 -14642.405,E2 -14642.405} C_VEL
LIN {X 0,Y 333.713,Z 227.913,A -85,B 0,C 180,E1 -14645.094,E2 -14645.094} C_VEL
LIN {X 0,Y 333.66,Z 227.92,A -85,B 0,C 180,E1 -14649.022,E2 -14649.022} C_VEL
LIN {X 0,Y 333.732,Z 227.914,A -85,B 0,C 180,E1 -14651.59,E2 -14651.59} C_VEL
LIN {X 0,Y 333.802,Z 227.907,A -85,B 0,C 180,E1 -14655.58,E2 -14655.58} C_VEL
LIN {X 0,Y 333.828,Z 227.9,A -85,B 0,C 180,E1 -14659.081,E2 -14659.081} C_VEL
LIN {X 0,Y 333.918,Z 227.962,A -85,B 0,C 180,E1 -14661.257,E2 -14661.257} C_VEL
LIN {X 0,Y 334.658,Z 231.77,A -85,B 0,C 180,E1 -14662.336,E2 -14662.336} C_VEL
LIN {X 0,Y 340.223,Z 249.273,A -85,B 0,C 180,E1 -14663.045,E2 -14663.045} C_VEL
LIN {X 0,Y 341.877,Z 258.747,A -85,B 0,C 180,E1 -14663.344,E2 -14663.344} C_VEL
LIN {X 0,Y 340.249,Z 339.488,A -85,B 0,C 180,E1 -14665.06,E2 -14665.06} C_VEL
LIN {X 0,Y 339.754,Z 352.856,A -85,B 0,C 180,E1 -14665.591,E2 -14665.591} C_VEL
LIN {X 0,Y 339.1,Z 364.801,A -85,B 0,C 180,E1 -14666.289,E2 -14666.289} C_VEL
LIN {X 0,Y 338.342,Z 376.103,A -85,B 0,C 180,E1 -14667.175,E2 -14667.175} C_VEL
LIN {X 0,Y 337.267,Z 388.072,A -85,B 0,C 180,E1 -14668.394,E2 -14668.394} C_VEL
LIN {X 0,Y 336.27,Z 398.27,A -85,B 0,C 180,E1 -14669.703,E2 -14669.703} C_VEL
LIN {X 0,Y 335.267,Z 407.725,A -85,B 0,C 180,E1 -14671.203,E2 -14671.203} C_VEL
LIN {X 0,Y 334.263,Z 416.829,A -85,B 0,C 180,E1 -14673.015,E2 -14673.015} C_VEL
LIN {X 0,Y 333.513,Z 424.163,A -85,B 0,C 180,E1 -14674.837,E2 -14674.837} C_VEL
LIN {X 0,Y 333.018,Z 429.793,A -85,B 0,C 180,E1 -14676.586,E2 -14676.586} C_VEL
LIN {X 0,Y 332.544,Z 434.67,A -85,B 0,C 180,E1 -14678.509,E2 -14678.509} C_VEL
LIN {X 0,Y 332.215,Z 438.2,A -85,B 0,C 180,E1 -14680.36,E2 -14680.36} C_VEL
LIN {X 0,Y 332.035,Z 440.705,A -85,B 0,C 180,E1 -14682.221,E2 -14682.221} C_VEL
LIN {X 0,Y 331.973,Z 441.823,A -85,B 0,C 180,E1 -14683.467,E2 -14683.467} C_VEL
LIN {X 0,Y 331.88,Z 442.532,A -85,B 0,C 180,E1 -14684.722,E2 -14684.722} C_VEL
LIN {X 0,Y 331.911,Z 442.839,A -85,B 0,C 180,E1 -14685.979,E2 -14685.979} C_VEL
LIN {X 0,Y 332.066,Z 442.531,A -85,B 0,C 180,E1 -14687.75,E2 -14687.75} C_VEL
LIN {X 0,Y 332.36,Z 441.169,A -85,B 0,C 180,E1 -14689.776,E2 -14689.776} C_VEL
LIN {X 0,Y 332.841,Z 438.812,A -85,B 0,C 180,E1 -14691.711,E2 -14691.711} C_VEL
LIN {X 0,Y 333.452,Z 435.447,A -85,B 0,C 180,E1 -14693.606,E2 -14693.606} C_VEL
LIN {X 0,Y 334.345,Z 430.568,A -85,B 0,C 180,E1 -14695.639,E2 -14695.639} C_VEL
LIN {X 0,Y 335.579,Z 423.793,A -85,B 0,C 180,E1 -14697.757,E2 -14697.757} C_VEL
LIN {X 0,Y 337.025,Z 415.89,A -85,B 0,C 180,E1 -14699.686,E2 -14699.686} C_VEL
LIN {X 0,Y 338.401,Z 407.737,A -85,B 0,C 180,E1 -14701.278,E2 -14701.278} C_VEL
LIN {X 0,Y 340.015,Z 397.621,A -85,B 0,C 180,E1 -14702.858,E2 -14702.858} C_VEL
LIN {X 0,Y 341.622,Z 386.921,A -85,B 0,C 180,E1 -14704.189,E2 -14704.189} C_VEL
LIN {X 0,Y 342.828,Z 376.729,A -85,B 0,C 180,E1 -14705.208,E2 -14705.208} C_VEL
LIN {X 0,Y 344.03,Z 364.577,A -85,B 0,C 180,E1 -14706.147,E2 -14706.147} C_VEL
LIN {X 0,Y 344.958,Z 352.185,A -85,B 0,C 180,E1 -14706.85,E2 -14706.85} C_VEL
LIN {X 0,Y 345.364,Z 344.494,A -85,B 0,C 180,E1 -14707.175,E2 -14707.175} C_VEL
LIN {X 0,Y 345.014,Z 338.759,A -85,B 0,C 180,E1 -14707.409,E2 -14707.409} C_VEL
LIN {X 0,Y 340.435,Z 320.177,A -85,B 0,C 180,E1 -14708.267,E2 -14708.267} C_VEL
LIN {X 0,Y 340.001,Z 314.383,A -85,B 0,C 180,E1 -14708.439,E2 -14708.439} C_VEL
LIN {X 0,Y 341.437,Z 263.193,A -85,B 0,C 180,E1 -14709.528,E2 -14709.528} C_VEL
LIN {X 0,Y 336.388,Z 251.026,A -85,B 0,C 180,E1 -14710.306,E2 -14710.306} C_VEL
LIN {X 0,Y 329.007,Z 235.79,A -85,B 0,C 180,E1 -14711.441,E2 -14711.441} C_VEL
LIN {X 0,Y 327.715,Z 233.001,A -85,B 0,C 180,E1 -14711.666,E2 -14711.666} C_VEL
LIN {X 0,Y 326.662,Z 228.8,A -85,B 0,C 180,E1 -14713.075,E2 -14713.075} C_VEL
LIN {X 0,Y 326.648,Z 228.8,A -85,B 0,C 180,E1 -14716.489,E2 -14716.489} C_VEL
LIN {X 0,Y 326.624,Z 228.796,A -85,B 0,C 180,E1 -14719.796,E2 -14719.796} C_VEL
LIN {X 0,Y 326.618,Z 228.798,A -85,B 0,C 180,E1 -14722.952,E2 -14722.952} C_VEL
LIN {X 0,Y 326.594,Z 228.8,A -85,B 0,C 180,E1 -14725.979,E2 -14725.979} C_VEL
LIN {X 0,Y 326.646,Z 228.792,A -85,B 0,C 180,E1 -14730.34,E2 -14730.34} C_VEL
LIN {X 0,Y 326.675,Z 228.784,A -85,B 0,C 180,E1 -14734.515,E2 -14734.515} C_VEL
LIN {X 0,Y 326.637,Z 228.787,A -85,B 0,C 180,E1 -14738.545,E2 -14738.545} C_VEL
LIN {X 0,Y 326.729,Z 228.785,A -85,B 0,C 180,E1 -14741.177,E2 -14741.177} C_VEL
LIN {X 0,Y 326.746,Z 228.786,A -85,B 0,C 180,E1 -14745.434,E2 -14745.434} C_VEL
LIN {X 0,Y 326.748,Z 228.78,A -85,B 0,C 180,E1 -14748.839,E2 -14748.839} C_VEL
LIN {X 0,Y 326.937,Z 228.75,A -85,B 0,C 180,E1 -14752.59,E2 -14752.59} C_VEL
LIN {X 0,Y 326.969,Z 228.754,A -85,B 0,C 180,E1 -14753.831,E2 -14753.831} C_VEL
LIN {X 0,Y 327.021,Z 228.741,A -85,B 0,C 180,E1 -14757.537,E2 -14757.537} C_VEL
LIN {X 0,Y 327.138,Z 228.726,A -85,B 0,C 180,E1 -14760,E2 -14760} C_VEL
LIN {X 0,Y 327.02,Z 228.74,A -85,B 0,C 180,E1 -14762.464,E2 -14762.464} C_VEL
LIN {X 0,Y 326.931,Z 228.746,A -85,B 0,C 180,E1 -14766.171,E2 -14766.171} C_VEL
LIN {X 0,Y 326.765,Z 228.767,A -85,B 0,C 180,E1 -14769.908,E2 -14769.908} C_VEL
LIN {X 0,Y 326.739,Z 228.776,A -85,B 0,C 180,E1 -14773.687,E2 -14773.687} C_VEL
LIN {X 0,Y 326.636,Z 228.793,A -85,B 0,C 180,E1 -14777.532,E2 -14777.532} C_VEL
LIN {X 0,Y 326.594,Z 228.801,A -85,B 0,C 180,E1 -14781.459,E2 -14781.459} C_VEL
LIN {X 0,Y 326.621,Z 228.799,A -85,B 0,C 180,E1 -14785.49,E2 -14785.49} C_VEL
LIN {X 0,Y 326.601,Z 228.801,A -85,B 0,C 180,E1 -14789.665,E2 -14789.665} C_VEL
LIN {X 0,Y 326.6,Z 228.802,A -85,B 0,C 180,E1 -14792.946,E2 -14792.946} C_VEL
LIN {X 0,Y 326.599,Z 228.801,A -85,B 0,C 180,E1 -14795.522,E2 -14795.522} C_VEL
LIN {X 0,Y 326.589,Z 228.804,A -85,B 0,C 180,E1 -14799.225,E2 -14799.225} C_VEL
LIN {X 0,Y 326.567,Z 228.797,A -85,B 0,C 180,E1 -14802.973,E2 -14802.973} C_VEL
LIN {X 0,Y 326.568,Z 228.805,A -85,B 0,C 180,E1 -14807.03,E2 -14807.03} C_VEL
LIN {X 0,Y 326.567,Z 228.8,A -85,B 0,C 180,E1 -14810.783,E2 -14810.783} C_VEL
LIN {X 0,Y 326.61,Z 228.805,A -85,B 0,C 180,E1 -14814.481,E2 -14814.481} C_VEL
LIN {X 0,Y 326.664,Z 229.008,A -85,B 0,C 180,E1 -14815.172,E2 -14815.172} C_VEL
LIN {X 0,Y 329.22,Z 238.956,A -85,B 0,C 180,E1 -14818.278,E2 -14818.278} C_VEL
LIN {X 0,Y 331.418,Z 248.779,A -85,B 0,C 180,E1 -14821.156,E2 -14821.156} C_VEL
LIN {X 0,Y 332.627,Z 255.961,A -85,B 0,C 180,E1 -14823.147,E2 -14823.147} C_VEL
LIN {X 0,Y 332.302,Z 259.25,A -85,B 0,C 180,E1 -14823.902,E2 -14823.902} C_VEL
LIN {X 0,Y 337.143,Z 282.056,A -85,B 0,C 180,E1 -14824.935,E2 -14824.935} C_VEL
LIN {X 0,Y 340.267,Z 301.246,A -85,B 0,C 180,E1 -14825.685,E2 -14825.685} C_VEL
LIN {X 0,Y 339.98,Z 320.058,A -85,B 0,C 180,E1 -14826.106,E2 -14826.106} C_VEL
LIN {X 0,Y 338.697,Z 368.688,A -85,B 0,C 180,E1 -14827.184,E2 -14827.184} C_VEL
LIN {X 0,Y 337.682,Z 382.373,A -85,B 0,C 180,E1 -14827.717,E2 -14827.717} C_VEL
LIN {X 0,Y 336.347,Z 395.225,A -85,B 0,C 180,E1 -14828.471,E2 -14828.471} C_VEL
LIN {X 0,Y 334.815,Z 406.942,A -85,B 0,C 180,E1 -14829.415,E2 -14829.415} C_VEL
LIN {X 0,Y 333.164,Z 418.252,A -85,B 0,C 180,E1 -14830.595,E2 -14830.595} C_VEL
LIN {X 0,Y 331.491,Z 428.487,A -85,B 0,C 180,E1 -14831.936,E2 -14831.936} C_VEL
LIN {X 0,Y 329.893,Z 437.859,A -85,B 0,C 180,E1 -14833.472,E2 -14833.472} C_VEL
LIN {X 0,Y 328.534,Z 446.032,A -85,B 0,C 180,E1 -14835.125,E2 -14835.125} C_VEL
LIN {X 0,Y 327.191,Z 453.425,A -85,B 0,C 180,E1 -14836.965,E2 -14836.965} C_VEL
LIN {X 0,Y 326.179,Z 459.385,A -85,B 0,C 180,E1 -14838.817,E2 -14838.817} C_VEL
LIN {X 0,Y 325.548,Z 464.119,A -85,B 0,C 180,E1 -14840.681,E2 -14840.681} C_VEL
LIN {X 0,Y 325.112,Z 467.759,A -85,B 0,C 180,E1 -14842.546,E2 -14842.546} C_VEL
LIN {X 0,Y 324.923,Z 470.215,A -85,B 0,C 180,E1 -14844.253,E2 -14844.253} C_VEL
LIN {X 0,Y 324.933,Z 472.125,A -85,B 0,C 180,E1 -14846.278,E2 -14846.278} C_VEL
LIN {X 0,Y 324.965,Z 473.033,A -85,B 0,C 180,E1 -14848.759,E2 -14848.759} C_VEL
LIN {X 0,Y 325.044,Z 472.862,A -85,B 0,C 180,E1 -14849.998,E2 -14849.998} C_VEL
LIN {X 0,Y 325.008,Z 472.283,A -85,B 0,C 180,E1 -14851.237,E2 -14851.237} C_VEL
LIN {X 0,Y 324.969,Z 469.93,A -85,B 0,C 180,E1 -14853.717,E2 -14853.717} C_VEL
LIN {X 0,Y 325.008,Z 466.398,A -85,B 0,C 180,E1 -14855.894,E2 -14855.894} C_VEL
LIN {X 0,Y 325.192,Z 461.405,A -85,B 0,C 180,E1 -14858.073,E2 -14858.073} C_VEL
LIN {X 0,Y 325.569,Z 455.824,A -85,B 0,C 180,E1 -14859.941,E2 -14859.941} C_VEL
LIN {X 0,Y 326.154,Z 448.838,A -85,B 0,C 180,E1 -14861.809,E2 -14861.809} C_VEL
LIN {X 0,Y 326.923,Z 441.7,A -85,B 0,C 180,E1 -14863.358,E2 -14863.358} C_VEL
LIN {X 0,Y 327.968,Z 431.987,A -85,B 0,C 180,E1 -14865.069,E2 -14865.069} C_VEL
LIN {X 0,Y 329.046,Z 421.176,A -85,B 0,C 180,E1 -14866.595,E2 -14866.595} C_VEL
LIN {X 0,Y 330.149,Z 410.28,A -85,B 0,C 180,E1 -14867.815,E2 -14867.815} C_VEL
LIN {X 0,Y 331.215,Z 399.043,A -85,B 0,C 180,E1 -14868.796,E2 -14868.796} C_VEL
LIN {X 0,Y 332.208,Z 386.544,A -85,B 0,C 180,E1 -14869.62,E2 -14869.62} C_VEL
LIN {X 0,Y 332.959,Z 373.61,A -85,B 0,C 180,E1 -14870.217,E2 -14870.217} C_VEL
LIN {X 0,Y 333.386,Z 359.818,A -85,B 0,C 180,E1 -14870.592,E2 -14870.592} C_VEL
LIN {X 0,Y 334.313,Z 299.523,A -85,B 0,C 180,E1 -14871.89,E2 -14871.89} C_VEL
LIN {X 0,Y 329.135,Z 259.923,A -85,B 0,C 180,E1 -14873.097,E2 -14873.097} C_VEL
LIN {X 0,Y 330.295,Z 248.27,A -85,B 0,C 180,E1 -14875.857,E2 -14875.857} C_VEL
LIN {X 0,Y 329.541,Z 242.617,A -85,B 0,C 180,E1 -14877.286,E2 -14877.286} C_VEL
LIN {X 0,Y 326.642,Z 228.795,A -85,B 0,C 180,E1 -14880.976,E2 -14880.976} C_VEL
LIN {X 0,Y 326.603,Z 228.8,A -85,B 0,C 180,E1 -14885.144,E2 -14885.144} C_VEL
LIN {X 0,Y 326.605,Z 228.8,A -85,B 0,C 180,E1 -14888.604,E2 -14888.604} C_VEL
LIN {X 0,Y 326.556,Z 228.81,A -85,B 0,C 180,E1 -14891.841,E2 -14891.841} C_VEL
LIN {X 0,Y 326.556,Z 228.806,A -85,B 0,C 180,E1 -14895.244,E2 -14895.244} C_VEL
LIN {X 0,Y 326.604,Z 228.799,A -85,B 0,C 180,E1 -14898.854,E2 -14898.854} C_VEL
LIN {X 0,Y 326.617,Z 228.8,A -85,B 0,C 180,E1 -14901.39,E2 -14901.39} C_VEL
LIN {X 0,Y 326.589,Z 228.801,A -85,B 0,C 180,E1 -14904.848,E2 -14904.848} C_VEL
LIN {X 0,Y 326.576,Z 228.806,A -85,B 0,C 180,E1 -14907.451,E2 -14907.451} C_VEL
LIN {X 0,Y 326.627,Z 228.796,A -85,B 0,C 180,E1 -14910.337,E2 -14910.337} C_VEL
LIN {X 0,Y 326.657,Z 228.792,A -85,B 0,C 180,E1 -14914.513,E2 -14914.513} C_VEL
LIN {X 0,Y 326.629,Z 228.796,A -85,B 0,C 180,E1 -14918.544,E2 -14918.544} C_VEL
LIN {X 0,Y 326.707,Z 228.789,A -85,B 0,C 180,E1 -14921.175,E2 -14921.175} C_VEL
LIN {X 0,Y 326.723,Z 228.788,A -85,B 0,C 180,E1 -14925.432,E2 -14925.432} C_VEL
LIN {X 0,Y 326.73,Z 228.784,A -85,B 0,C 180,E1 -14928.837,E2 -14928.837} C_VEL
LIN {X 0,Y 326.942,Z 228.757,A -85,B 0,C 180,E1 -14932.589,E2 -14932.589} C_VEL
LIN {X 0,Y 326.736,Z 228.787,A -85,B 0,C 180,E1 -14935.064,E2 -14935.064} C_VEL
LIN {X 0,Y 327.001,Z 228.748,A -85,B 0,C 180,E1 -14937.536,E2 -14937.536} C_VEL
LIN {X 0,Y 327.133,Z 228.728,A -85,B 0,C 180,E1 -14940,E2 -14940} C_VEL
LIN {X 0,Y 326.998,Z 228.748,A -85,B 0,C 180,E1 -14942.463,E2 -14942.463} C_VEL
LIN {X 0,Y 326.909,Z 228.759,A -85,B 0,C 180,E1 -14946.714,E2 -14946.714} C_VEL
LIN {X 0,Y 326.763,Z 228.778,A -85,B 0,C 180,E1 -14949.907,E2 -14949.907} C_VEL
LIN {X 0,Y 326.715,Z 228.785,A -85,B 0,C 180,E1 -14953.687,E2 -14953.687} C_VEL
LIN {X 0,Y 326.632,Z 228.795,A -85,B 0,C 180,E1 -14957.531,E2 -14957.531} C_VEL
LIN {X 0,Y 326.571,Z 228.803,A -85,B 0,C 180,E1 -14961.459,E2 -14961.459} C_VEL
LIN {X 0,Y 326.634,Z 228.794,A -85,B 0,C 180,E1 -14965.488,E2 -14965.488} C_VEL
LIN {X 0,Y 326.606,Z 228.799,A -85,B 0,C 180,E1 -14968.255,E2 -14968.255} C_VEL
LIN {X 0,Y 326.536,Z 228.804,A -85,B 0,C 180,E1 -14971.101,E2 -14971.101} C_VEL
LIN {X 0,Y 326.573,Z 228.802,A -85,B 0,C 180,E1 -14974.023,E2 -14974.023} C_VEL
LIN {X 0,Y 326.595,Z 228.8,A -85,B 0,C 180,E1 -14977.241,E2 -14977.241} C_VEL
LIN {X 0,Y 326.548,Z 228.804,A -85,B 0,C 180,E1 -14981.135,E2 -14981.135} C_VEL
LIN {X 0,Y 326.5,Z 228.813,A -85,B 0,C 180,E1 -14984.746,E2 -14984.746} C_VEL
LIN {X 0,Y 326.552,Z 228.81,A -85,B 0,C 180,E1 -14988.158,E2 -14988.158} C_VEL
LIN {X 0,Y 326.576,Z 228.801,A -85,B 0,C 180,E1 -14991.392,E2 -14991.392} C_VEL
LIN {X 0,Y 326.6,Z 228.8,A -85,B 0,C 180,E1 -14994.856,E2 -14994.856} C_VEL
LIN {X 0,Y 326.59,Z 228.801,A -85,B 0,C 180,E1 -14997.459,E2 -14997.459} C_VEL
LIN {X 0,Y 326.632,Z 228.798,A -85,B 0,C 180,E1 -15000.344,E2 -15000.344} C_VEL
LIN {X 0,Y 326.677,Z 228.791,A -85,B 0,C 180,E1 -15004.52,E2 -15004.52} C_VEL
LIN {X 0,Y 326.607,Z 228.799,A -85,B 0,C 180,E1 -15008.547,E2 -15008.547} C_VEL
LIN {X 0,Y 326.655,Z 228.794,A -85,B 0,C 180,E1 -15012.474,E2 -15012.474} C_VEL
LIN {X 0,Y 326.753,Z 228.783,A -85,B 0,C 180,E1 -15016.318,E2 -15016.318} C_VEL
LIN {X 0,Y 326.799,Z 228.777,A -85,B 0,C 180,E1 -15020.096,E2 -15020.096} C_VEL
LIN {X 0,Y 326.861,Z 228.889,A -85,B 0,C 180,E1 -15020.981,E2 -15020.981} C_VEL
LIN {X 0,Y 327.524,Z 232.126,A -85,B 0,C 180,E1 -15021.92,E2 -15021.92} C_VEL
LIN {X 0,Y 333.604,Z 250.781,A -85,B 0,C 180,E1 -15022.703,E2 -15022.703} C_VEL
LIN {X 0,Y 335.106,Z 258.664,A -85,B 0,C 180,E1 -15022.967,E2 -15022.967} C_VEL
LIN {X 0,Y 333.449,Z 339.384,A -85,B 0,C 180,E1 -15024.712,E2 -15024.712} C_VEL
LIN {X 0,Y 332.969,Z 352.518,A -85,B 0,C 180,E1 -15025.235,E2 -15025.235} C_VEL
LIN {X 0,Y 332.24,Z 365.203,A -85,B 0,C 180,E1 -15025.984,E2 -15025.984} C_VEL
LIN {X 0,Y 331.393,Z 377.275,A -85,B 0,C 180,E1 -15026.963,E2 -15026.963} C_VEL
LIN {X 0,Y 330.376,Z 388.274,A -85,B 0,C 180,E1 -15028.113,E2 -15028.113} C_VEL
LIN {X 0,Y 329.288,Z 399.159,A -85,B 0,C 180,E1 -15029.544,E2 -15029.544} C_VEL
LIN {X 0,Y 328.332,Z 407.649,A -85,B 0,C 180,E1 -15030.922,E2 -15030.922} C_VEL
LIN {X 0,Y 327.282,Z 416.836,A -85,B 0,C 180,E1 -15032.771,E2 -15032.771} C_VEL
LIN {X 0,Y 326.489,Z 424.228,A -85,B 0,C 180,E1 -15034.632,E2 -15034.632} C_VEL
LIN {X 0,Y 326.031,Z 429.236,A -85,B 0,C 180,E1 -15036.189,E2 -15036.189} C_VEL
LIN {X 0,Y 325.562,Z 434.11,A -85,B 0,C 180,E1 -15038.068,E2 -15038.068} C_VEL
LIN {X 0,Y 325.199,Z 437.86,A -85,B 0,C 180,E1 -15039.957,E2 -15039.957} C_VEL
LIN {X 0,Y 325.03,Z 439.801,A -85,B 0,C 180,E1 -15041.223,E2 -15041.223} C_VEL
LIN {X 0,Y 324.917,Z 441.967,A -85,B 0,C 180,E1 -15043.257,E2 -15043.257} C_VEL
LIN {X 0,Y 324.797,Z 442.96,A -85,B 0,C 180,E1 -15045.051,E2 -15045.051} C_VEL
LIN {X 0,Y 324.859,Z 443.189,A -85,B 0,C 180,E1 -15046.335,E2 -15046.335} C_VEL
LIN {X 0,Y 325.007,Z 442.851,A -85,B 0,C 180,E1 -15047.926,E2 -15047.926} C_VEL
LIN {X 0,Y 325.358,Z 441.279,A -85,B 0,C 180,E1 -15050.22,E2 -15050.22} C_VEL
LIN {X 0,Y 325.817,Z 439.14,A -85,B 0,C 180,E1 -15051.949,E2 -15051.949} C_VEL
LIN {X 0,Y 326.582,Z 435.276,A -85,B 0,C 180,E1 -15054.134,E2 -15054.134} C_VEL
LIN {X 0,Y 327.508,Z 430.503,A -85,B 0,C 180,E1 -15056.097,E2 -15056.097} C_VEL
LIN {X 0,Y 328.7,Z 424.333,A -85,B 0,C 180,E1 -15058.059,E2 -15058.059} C_VEL
LIN {X 0,Y 330.212,Z 416.546,A -85,B 0,C 180,E1 -15060.01,E2 -15060.01} C_VEL
LIN {X 0,Y 331.661,Z 408.491,A -85,B 0,C 180,E1 -15061.631,E2 -15061.631} C_VEL
LIN {X 0,Y 333.351,Z 398.493,A -85,B 0,C 180,E1 -15063.24,E2 -15063.24} C_VEL
LIN {X 0,Y 334.924,Z 388.631,A -85,B 0,C 180,E1 -15064.51,E2 -15064.51} C_VEL
LIN {X 0,Y 336.294,Z 377.923,A -85,B 0,C 180,E1 -15065.626,E2 -15065.626} C_VEL
LIN {X 0,Y 337.543,Z 366.105,A -85,B 0,C 180,E1 -15066.583,E2 -15066.583} C_VEL
LIN {X 0,Y 338.539,Z 353.467,A -85,B 0,C 180,E1 -15067.332,E2 -15067.332} C_VEL
LIN {X 0,Y 339.229,Z 340.801,A -85,B 0,C 180,E1 -15067.841,E2 -15067.841} C_VEL
LIN {X 0,Y 340.001,Z 314.383,A -85,B 0,C 180,E1 -15068.439,E2 -15068.439} C_VEL
LIN {X 0,Y 339.584,Z 308.587,A -85,B 0,C 180,E1 -15068.615,E2 -15068.615} C_VEL
LIN {X 0,Y 335.112,Z 289.955,A -85,B 0,C 180,E1 -15069.479,E2 -15069.479} C_VEL
LIN {X 0,Y 334.617,Z 284.163,A -85,B 0,C 180,E1 -15069.668,E2 -15069.668} C_VEL
LIN {X 0,Y 335.084,Z 264.556,A -85,B 0,C 180,E1 -15070.103,E2 -15070.103} C_VEL
LIN {X 0,Y 327.378,Z 246.941,A -85,B 0,C 180,E1 -15071.33,E2 -15071.33} C_VEL
LIN {X 0,Y 320.531,Z 233.411,A -85,B 0,C 180,E1 -15072.444,E2 -15072.444} C_VEL
LIN {X 0,Y 319.596,Z 229.677,A -85,B 0,C 180,E1 -15073.729,E2 -15073.729} C_VEL
LIN {X 0,Y 319.616,Z 229.673,A -85,B 0,C 180,E1 -15077.027,E2 -15077.027} C_VEL
LIN {X 0,Y 319.573,Z 229.676,A -85,B 0,C 180,E1 -15080.375,E2 -15080.375} C_VEL
LIN {X 0,Y 319.546,Z 229.681,A -85,B 0,C 180,E1 -15083.571,E2 -15083.571} C_VEL
LIN {X 0,Y 319.565,Z 229.677,A -85,B 0,C 180,E1 -15086.686,E2 -15086.686} C_VEL
LIN {X 0,Y 319.578,Z 229.675,A -85,B 0,C 180,E1 -15089.616,E2 -15089.616} C_VEL
LIN {X 0,Y 319.594,Z 229.671,A -85,B 0,C 180,E1 -15092.497,E2 -15092.497} C_VEL
LIN {X 0,Y 319.59,Z 229.665,A -85,B 0,C 180,E1 -15095.303,E2 -15095.303} C_VEL
LIN {X 0,Y 319.584,Z 229.668,A -85,B 0,C 180,E1 -15098.047,E2 -15098.047} C_VEL
LIN {X 0,Y 319.674,Z 229.663,A -85,B 0,C 180,E1 -15100.962,E2 -15100.962} C_VEL
LIN {X 0,Y 319.714,Z 229.661,A -85,B 0,C 180,E1 -15105.277,E2 -15105.277} C_VEL
LIN {X 0,Y 319.733,Z 229.657,A -85,B 0,C 180,E1 -15109.872,E2 -15109.872} C_VEL
LIN {X 0,Y 319.923,Z 229.633,A -85,B 0,C 180,E1 -15113.694,E2 -15113.694} C_VEL
LIN {X 0,Y 319.965,Z 229.619,A -85,B 0,C 180,E1 -15117.483,E2 -15117.483} C_VEL
LIN {X 0,Y 320.092,Z 229.603,A -85,B 0,C 180,E1 -15120,E2 -15120} C_VEL
LIN {X 0,Y 319.964,Z 229.619,A -85,B 0,C 180,E1 -15122.518,E2 -15122.518} C_VEL
LIN {X 0,Y 319.888,Z 229.624,A -85,B 0,C 180,E1 -15126.307,E2 -15126.307} C_VEL
LIN {X 0,Y 319.718,Z 229.645,A -85,B 0,C 180,E1 -15130.129,E2 -15130.129} C_VEL
LIN {X 0,Y 319.714,Z 229.651,A -85,B 0,C 180,E1 -15133.993,E2 -15133.993} C_VEL
LIN {X 0,Y 319.584,Z 229.671,A -85,B 0,C 180,E1 -15137.932,E2 -15137.932} C_VEL
LIN {X 0,Y 319.549,Z 229.678,A -85,B 0,C 180,E1 -15141.956,E2 -15141.956} C_VEL
LIN {X 0,Y 319.556,Z 229.679,A -85,B 0,C 180,E1 -15146.095,E2 -15146.095} C_VEL
LIN {X 0,Y 319.529,Z 229.685,A -85,B 0,C 180,E1 -15148.94,E2 -15148.94} C_VEL
LIN {X 0,Y 319.506,Z 229.681,A -85,B 0,C 180,E1 -15151.865,E2 -15151.865} C_VEL
LIN {X 0,Y 319.567,Z 229.677,A -85,B 0,C 180,E1 -15155.543,E2 -15155.543} C_VEL
LIN {X 0,Y 319.552,Z 229.681,A -85,B 0,C 180,E1 -15159.67,E2 -15159.67} C_VEL
LIN {X 0,Y 319.513,Z 229.683,A -85,B 0,C 180,E1 -15163.461,E2 -15163.461} C_VEL
LIN {X 0,Y 319.546,Z 229.68,A -85,B 0,C 180,E1 -15167.017,E2 -15167.017} C_VEL
LIN {X 0,Y 319.511,Z 229.677,A -85,B 0,C 180,E1 -15170.367,E2 -15170.367} C_VEL
LIN {X 0,Y 319.594,Z 229.748,A -85,B 0,C 180,E1 -15174.454,E2 -15174.454} C_VEL
LIN {X 0,Y 322.156,Z 239.745,A -85,B 0,C 180,E1 -15177.681,E2 -15177.681} C_VEL
LIN {X 0,Y 324.252,Z 248.835,A -85,B 0,C 180,E1 -15180.439,E2 -15180.439} C_VEL
LIN {X 0,Y 325.677,Z 256.072,A -85,B 0,C 180,E1 -15182.527,E2 -15182.527} C_VEL
LIN {X 0,Y 325.722,Z 258.593,A -85,B 0,C 180,E1 -15183.199,E2 -15183.199} C_VEL
LIN {X 0,Y 330.416,Z 280.622,A -85,B 0,C 180,E1 -15184.245,E2 -15184.245} C_VEL
LIN {X 0,Y 333.597,Z 299.308,A -85,B 0,C 180,E1 -15185.017,E2 -15185.017} C_VEL
LIN {X 0,Y 334.12,Z 304.338,A -85,B 0,C 180,E1 -15185.189,E2 -15185.189} C_VEL
LIN {X 0,Y 332.425,Z 367.75,A -85,B 0,C 180,E1 -15186.605,E2 -15186.605} C_VEL
LIN {X 0,Y 331.466,Z 380.873,A -85,B 0,C 180,E1 -15187.112,E2 -15187.112} C_VEL
LIN {X 0,Y 330.092,Z 394.08,A -85,B 0,C 180,E1 -15187.878,E2 -15187.878} C_VEL
LIN {X 0,Y 328.487,Z 406,A -85,B 0,C 180,E1 -15188.836,E2 -15188.836} C_VEL
LIN {X 0,Y 326.699,Z 417.425,A -85,B 0,C 180,E1 -15190.031,E2 -15190.031} C_VEL
LIN {X 0,Y 324.931,Z 427.749,A -85,B 0,C 180,E1 -15191.395,E2 -15191.395} C_VEL
LIN {X 0,Y 323.197,Z 437.39,A -85,B 0,C 180,E1 -15192.993,E2 -15192.993} C_VEL
LIN {X 0,Y 321.655,Z 446.103,A -85,B 0,C 180,E1 -15194.799,E2 -15194.799} C_VEL
LIN {X 0,Y 320.277,Z 453.42,A -85,B 0,C 180,E1 -15196.678,E2 -15196.678} C_VEL
LIN {X 0,Y 319.169,Z 459.314,A -85,B 0,C 180,E1 -15198.568,E2 -15198.568} C_VEL
LIN {X 0,Y 318.503,Z 463.992,A -85,B 0,C 180,E1 -15200.473,E2 -15200.473} C_VEL
LIN {X 0,Y 318.035,Z 467.58,A -85,B 0,C 180,E1 -15202.379,E2 -15202.379} C_VEL
LIN {X 0,Y 317.841,Z 470.178,A -85,B 0,C 180,E1 -15204.286,E2 -15204.286} C_VEL
LIN {X 0,Y 317.837,Z 471.852,A -85,B 0,C 180,E1 -15206.195,E2 -15206.195} C_VEL
LIN {X 0,Y 317.814,Z 472.477,A -85,B 0,C 180,E1 -15207.463,E2 -15207.463} C_VEL
LIN {X 0,Y 317.868,Z 472.704,A -85,B 0,C 180,E1 -15208.731,E2 -15208.731} C_VEL
LIN {X 0,Y 317.953,Z 472.499,A -85,B 0,C 180,E1 -15209.998,E2 -15209.998} C_VEL
LIN {X 0,Y 317.912,Z 471.897,A -85,B 0,C 180,E1 -15211.264,E2 -15211.264} C_VEL
LIN {X 0,Y 317.846,Z 470.897,A -85,B 0,C 180,E1 -15212.532,E2 -15212.532} C_VEL
LIN {X 0,Y 317.897,Z 469.487,A -85,B 0,C 180,E1 -15213.8,E2 -15213.8} C_VEL
LIN {X 0,Y 317.911,Z 466.26,A -85,B 0,C 180,E1 -15215.838,E2 -15215.838} C_VEL
LIN {X 0,Y 318.044,Z 462.468,A -85,B 0,C 180,E1 -15217.616,E2 -15217.616} C_VEL
LIN {X 0,Y 318.456,Z 456.225,A -85,B 0,C 180,E1 -15219.845,E2 -15219.845} C_VEL
LIN {X 0,Y 319.017,Z 449.4,A -85,B 0,C 180,E1 -15221.755,E2 -15221.755} C_VEL
LIN {X 0,Y 319.935,Z 440.917,A -85,B 0,C 180,E1 -15223.656,E2 -15223.656} C_VEL
LIN {X 0,Y 320.937,Z 432.159,A -85,B 0,C 180,E1 -15225.231,E2 -15225.231} C_VEL
LIN {X 0,Y 322.063,Z 421.35,A -85,B 0,C 180,E1 -15226.803,E2 -15226.803} C_VEL
LIN {X 0,Y 323.188,Z 410.599,A -85,B 0,C 180,E1 -15228.048,E2 -15228.048} C_VEL
LIN {X 0,Y 324.387,Z 398.56,A -85,B 0,C 180,E1 -15229.125,E2 -15229.125} C_VEL
LIN {X 0,Y 325.399,Z 386.011,A -85,B 0,C 180,E1 -15229.965,E2 -15229.965} C_VEL
LIN {X 0,Y 326.179,Z 372.938,A -85,B 0,C 180,E1 -15230.573,E2 -15230.573} C_VEL
LIN {X 0,Y 326.65,Z 357.137,A -85,B 0,C 180,E1 -15230.996,E2 -15230.996} C_VEL
LIN {X 0,Y 327.594,Z 300.517,A -85,B 0,C 180,E1 -15232.237,E2 -15232.237} C_VEL
LIN {X 0,Y 322.231,Z 259.659,A -85,B 0,C 180,E1 -15233.499,E2 -15233.499} C_VEL
LIN {X 0,Y 323.305,Z 249.048,A -85,B 0,C 180,E1 -15236.07,E2 -15236.07} C_VEL
LIN {X 0,Y 322.14,Z 241.781,A -85,B 0,C 180,E1 -15237.968,E2 -15237.968} C_VEL
LIN {X 0,Y 319.56,Z 229.678,A -85,B 0,C 180,E1 -15241.285,E2 -15241.285} C_VEL
LIN {X 0,Y 319.544,Z 229.68,A -85,B 0,C 180,E1 -15244.872,E2 -15244.872} C_VEL
LIN {X 0,Y 319.555,Z 229.683,A -85,B 0,C 180,E1 -15248.004,E2 -15248.004} C_VEL
LIN {X 0,Y 319.506,Z 229.686,A -85,B 0,C 180,E1 -15251.592,E2 -15251.592} C_VEL
LIN {X 0,Y 319.536,Z 229.68,A -85,B 0,C 180,E1 -15255.265,E2 -15255.265} C_VEL
LIN {X 0,Y 319.554,Z 229.677,A -85,B 0,C 180,E1 -15258.715,E2 -15258.715} C_VEL
LIN {X 0,Y 319.554,Z 229.678,A -85,B 0,C 180,E1 -15262.339,E2 -15262.339} C_VEL
LIN {X 0,Y 319.529,Z 229.681,A -85,B 0,C 180,E1 -15265.119,E2 -15265.119} C_VEL
LIN {X 0,Y 319.538,Z 229.68,A -85,B 0,C 180,E1 -15269.055,E2 -15269.055} C_VEL
LIN {X 0,Y 319.574,Z 229.674,A -85,B 0,C 180,E1 -15272.494,E2 -15272.494} C_VEL
LIN {X 0,Y 319.576,Z 229.678,A -85,B 0,C 180,E1 -15275.301,E2 -15275.301} C_VEL
LIN {X 0,Y 319.595,Z 229.677,A -85,B 0,C 180,E1 -15279.399,E2 -15279.399} C_VEL
LIN {X 0,Y 319.619,Z 229.668,A -85,B 0,C 180,E1 -15282.07,E2 -15282.07} C_VEL
LIN {X 0,Y 319.691,Z 229.66,A -85,B 0,C 180,E1 -15286.006,E2 -15286.006} C_VEL
LIN {X 0,Y 319.718,Z 229.657,A -85,B 0,C 180,E1 -15289.871,E2 -15289.871} C_VEL
LIN {X 0,Y 319.895,Z 229.635,A -85,B 0,C 180,E1 -15292.425,E2 -15292.425} C_VEL
LIN {X 0,Y 319.706,Z 229.661,A -85,B 0,C 180,E1 -15294.955,E2 -15294.955} C_VEL
LIN {X 0,Y 319.945,Z 229.626,A -85,B 0,C 180,E1 -15297.482,E2 -15297.482} C_VEL
LIN {X 0,Y 320.086,Z 229.604,A -85,B 0,C 180,E1 -15300,E2 -15300} C_VEL
LIN {X 0,Y 319.942,Z 229.626,A -85,B 0,C 180,E1 -15302.518,E2 -15302.518} C_VEL
LIN {X 0,Y 319.869,Z 229.636,A -85,B 0,C 180,E1 -15306.703,E2 -15306.703} C_VEL
LIN {X 0,Y 319.71,Z 229.657,A -85,B 0,C 180,E1 -15310.128,E2 -15310.128} C_VEL
LIN {X 0,Y 319.689,Z 229.66,A -85,B 0,C 180,E1 -15313.994,E2 -15313.994} C_VEL
LIN {X 0,Y 319.58,Z 229.673,A -85,B 0,C 180,E1 -15317.931,E2 -15317.931} C_VEL
LIN {X 0,Y 319.526,Z 229.68,A -85,B 0,C 180,E1 -15321.957,E2 -15321.957} C_VEL
LIN {X 0,Y 319.571,Z 229.675,A -85,B 0,C 180,E1 -15326.093,E2 -15326.093} C_VEL
LIN {X 0,Y 319.528,Z 229.677,A -85,B 0,C 180,E1 -15328.939,E2 -15328.939} C_VEL
LIN {X 0,Y 319.488,Z 229.68,A -85,B 0,C 180,E1 -15331.866,E2 -15331.866} C_VEL
LIN {X 0,Y 319.546,Z 229.677,A -85,B 0,C 180,E1 -15335.546,E2 -15335.546} C_VEL
LIN {X 0,Y 319.526,Z 229.682,A -85,B 0,C 180,E1 -15338.014,E2 -15338.014} C_VEL
LIN {X 0,Y 319.497,Z 229.682,A -85,B 0,C 180,E1 -15341.6,E2 -15341.6} C_VEL
LIN {X 0,Y 319.461,Z 229.687,A -85,B 0,C 180,E1 -15345.261,E2 -15345.261} C_VEL
LIN {X 0,Y 319.505,Z 229.685,A -85,B 0,C 180,E1 -15348.716,E2 -15348.716} C_VEL
LIN {X 0,Y 319.533,Z 229.681,A -85,B 0,C 180,E1 -15352.354,E2 -15352.354} C_VEL
LIN {X 0,Y 319.541,Z 229.678,A -85,B 0,C 180,E1 -15355.127,E2 -15355.127} C_VEL
LIN {X 0,Y 319.55,Z 229.676,A -85,B 0,C 180,E1 -15359.063,E2 -15359.063} C_VEL
LIN {X 0,Y 319.591,Z 229.674,A -85,B 0,C 180,E1 -15362.502,E2 -15362.502} C_VEL
LIN {X 0,Y 319.59,Z 229.673,A -85,B 0,C 180,E1 -15365.308,E2 -15365.308} C_VEL
LIN {X 0,Y 319.572,Z 229.677,A -85,B 0,C 180,E1 -15369.403,E2 -15369.403} C_VEL
LIN {X 0,Y 319.649,Z 229.668,A -85,B 0,C 180,E1 -15373.396,E2 -15373.396} C_VEL
LIN {X 0,Y 319.726,Z 229.661,A -85,B 0,C 180,E1 -15376.011,E2 -15376.011} C_VEL
LIN {X 0,Y 319.747,Z 229.658,A -85,B 0,C 180,E1 -15379.876,E2 -15379.876} C_VEL
LIN {X 0,Y 319.792,Z 229.775,A -85,B 0,C 180,E1 -15380.692,E2 -15380.692} C_VEL
LIN {X 0,Y 320.352,Z 232.341,A -85,B 0,C 180,E1 -15381.454,E2 -15381.454} C_VEL
LIN {X 0,Y 326.798,Z 251.747,A -85,B 0,C 180,E1 -15382.328,E2 -15382.328} C_VEL
LIN {X 0,Y 328.344,Z 259.586,A -85,B 0,C 180,E1 -15382.599,E2 -15382.599} C_VEL
LIN {X 0,Y 326.646,Z 339.824,A -85,B 0,C 180,E1 -15384.369,E2 -15384.369} C_VEL
LIN {X 0,Y 326.15,Z 352.922,A -85,B 0,C 180,E1 -15384.903,E2 -15384.903} C_VEL
LIN {X 0,Y 325.39,Z 365.594,A -85,B 0,C 180,E1 -15385.667,E2 -15385.667} C_VEL
LIN {X 0,Y 324.581,Z 376.808,A -85,B 0,C 180,E1 -15386.584,E2 -15386.584} C_VEL
LIN {X 0,Y 323.528,Z 388.183,A -85,B 0,C 180,E1 -15387.785,E2 -15387.785} C_VEL
LIN {X 0,Y 322.383,Z 398.987,A -85,B 0,C 180,E1 -15389.222,E2 -15389.222} C_VEL
LIN {X 0,Y 321.42,Z 407.554,A -85,B 0,C 180,E1 -15390.629,E2 -15390.629} C_VEL
LIN {X 0,Y 320.473,Z 415.46,A -85,B 0,C 180,E1 -15392.201,E2 -15392.201} C_VEL
LIN {X 0,Y 319.627,Z 423.163,A -85,B 0,C 180,E1 -15394.1,E2 -15394.1} C_VEL
LIN {X 0,Y 319.031,Z 428.444,A -85,B 0,C 180,E1 -15395.691,E2 -15395.691} C_VEL
LIN {X 0,Y 318.582,Z 433.544,A -85,B 0,C 180,E1 -15397.608,E2 -15397.608} C_VEL
LIN {X 0,Y 318.166,Z 437.518,A -85,B 0,C 180,E1 -15399.537,E2 -15399.537} C_VEL
LIN {X 0,Y 317.913,Z 440.441,A -85,B 0,C 180,E1 -15401.477,E2 -15401.477} C_VEL
LIN {X 0,Y 317.814,Z 442.325,A -85,B 0,C 180,E1 -15403.347,E2 -15403.347} C_VEL
LIN {X 0,Y 317.72,Z 443.379,A -85,B 0,C 180,E1 -15405.394,E2 -15405.394} C_VEL
LIN {X 0,Y 317.793,Z 443.493,A -85,B 0,C 180,E1 -15406.709,E2 -15406.709} C_VEL
LIN {X 0,Y 317.952,Z 443.171,A -85,B 0,C 180,E1 -15408.11,E2 -15408.11} C_VEL
LIN {X 0,Y 318.11,Z 442.503,A -85,B 0,C 180,E1 -15409.354,E2 -15409.354} C_VEL
LIN {X 0,Y 318.373,Z 441.34,A -85,B 0,C 180,E1 -15410.683,E2 -15410.683} C_VEL
LIN {X 0,Y 318.836,Z 439.444,A -85,B 0,C 180,E1 -15412.213,E2 -15412.213} C_VEL
LIN {X 0,Y 319.454,Z 436.405,A -85,B 0,C 180,E1 -15414.017,E2 -15414.017} C_VEL
LIN {X 0,Y 320.388,Z 431.908,A -85,B 0,C 180,E1 -15416.022,E2 -15416.022} C_VEL
LIN {X 0,Y 321.635,Z 426.088,A -85,B 0,C 180,E1 -15418.02,E2 -15418.02} C_VEL
LIN {X 0,Y 323.134,Z 418.647,A -85,B 0,C 180,E1 -15420.015,E2 -15420.015} C_VEL
LIN {X 0,Y 324.617,Z 410.96,A -85,B 0,C 180,E1 -15421.669,E2 -15421.669} C_VEL
LIN {X 0,Y 326.26,Z 401.946,A -85,B 0,C 180,E1 -15423.244,E2 -15423.244} C_VEL
LIN {X 0,Y 327.876,Z 392.283,A -85,B 0,C 180,E1 -15424.612,E2 -15424.612} C_VEL
LIN {X 0,Y 329.52,Z 381.186,A -85,B 0,C 180,E1 -15425.859,E2 -15425.859} C_VEL
LIN {X 0,Y 330.877,Z 369.672,A -85,B 0,C 180,E1 -15426.872,E2 -15426.872} C_VEL
LIN {X 0,Y 331.931,Z 357.481,A -85,B 0,C 180,E1 -15427.687,E2 -15427.687} C_VEL
LIN {X 0,Y 332.771,Z 344.299,A -85,B 0,C 180,E1 -15428.292,E2 -15428.292} C_VEL
LIN {X 0,Y 333.33,Z 326.835,A -85,B 0,C 180,E1 -15428.749,E2 -15428.749} C_VEL
LIN {X 0,Y 334.617,Z 284.163,A -85,B 0,C 180,E1 -15429.668,E2 -15429.668} C_VEL
LIN {X 0,Y 333.994,Z 279.03,A -85,B 0,C 180,E1 -15429.854,E2 -15429.854} C_VEL
LIN {X 0,Y 332.423,Z 274.197,A -85,B 0,C 180,E1 -15430.128,E2 -15430.128} C_VEL
LIN {X 0,Y 328.282,Z 264.874,A -85,B 0,C 180,E1 -15430.781,E2 -15430.781} C_VEL
LIN {X 0,Y 320.759,Z 248.076,A -85,B 0,C 180,E1 -15432.021,E2 -15432.021} C_VEL
LIN {X 0,Y 313.373,Z 233.818,A -85,B 0,C 180,E1 -15433.267,E2 -15433.267} C_VEL
LIN {X 0,Y 312.569,Z 230.554,A -85,B 0,C 180,E1 -15434.428,E2 -15434.428} C_VEL
LIN {X 0,Y 312.547,Z 230.551,A -85,B 0,C 180,E1 -15437.903,E2 -15437.903} C_VEL
LIN {X 0,Y 312.532,Z 230.552,A -85,B 0,C 180,E1 -15441.908,E2 -15441.908} C_VEL
LIN {X 0,Y 312.494,Z 230.554,A -85,B 0,C 180,E1 -15445.789,E2 -15445.789} C_VEL
LIN {X 0,Y 312.51,Z 230.552,A -85,B 0,C 180,E1 -15448.853,E2 -15448.853} C_VEL
LIN {X 0,Y 312.56,Z 230.542,A -85,B 0,C 180,E1 -15451.824,E2 -15451.824} C_VEL
LIN {X 0,Y 312.571,Z 230.54,A -85,B 0,C 180,E1 -15454.71,E2 -15454.71} C_VEL
LIN {X 0,Y 312.573,Z 230.547,A -85,B 0,C 180,E1 -15457.528,E2 -15457.528} C_VEL
LIN {X 0,Y 312.622,Z 230.541,A -85,B 0,C 180,E1 -15461.656,E2 -15461.656} C_VEL
LIN {X 0,Y 312.675,Z 230.536,A -85,B 0,C 180,E1 -15465.686,E2 -15465.686} C_VEL
LIN {X 0,Y 312.679,Z 230.537,A -85,B 0,C 180,E1 -15469.641,E2 -15469.641} C_VEL
LIN {X 0,Y 312.827,Z 230.507,A -85,B 0,C 180,E1 -15472.254,E2 -15472.254} C_VEL
LIN {X 0,Y 312.88,Z 230.508,A -85,B 0,C 180,E1 -15473.552,E2 -15473.552} C_VEL
LIN {X 0,Y 312.912,Z 230.497,A -85,B 0,C 180,E1 -15477.426,E2 -15477.426} C_VEL
LIN {X 0,Y 313.047,Z 230.481,A -85,B 0,C 180,E1 -15480,E2 -15480} C_VEL
LIN {X 0,Y 312.911,Z 230.498,A -85,B 0,C 180,E1 -15482.575,E2 -15482.575} C_VEL
LIN {X 0,Y 312.83,Z 230.503,A -85,B 0,C 180,E1 -15486.45,E2 -15486.45} C_VEL
LIN {X 0,Y 312.734,Z 230.52,A -85,B 0,C 180,E1 -15489.051,E2 -15489.051} C_VEL
LIN {X 0,Y 312.616,Z 230.54,A -85,B 0,C 180,E1 -15492.992,E2 -15492.992} C_VEL
LIN {X 0,Y 312.604,Z 230.538,A -85,B 0,C 180,E1 -15495.652,E2 -15495.652} C_VEL
LIN {X 0,Y 312.52,Z 230.548,A -85,B 0,C 180,E1 -15499.714,E2 -15499.714} C_VEL
LIN {X 0,Y 312.507,Z 230.551,A -85,B 0,C 180,E1 -15502.779,E2 -15502.779} C_VEL
LIN {X 0,Y 312.516,Z 230.556,A -85,B 0,C 180,E1 -15505.908,E2 -15505.908} C_VEL
LIN {X 0,Y 312.482,Z 230.56,A -85,B 0,C 180,E1 -15509.657,E2 -15509.657} C_VEL
LIN {X 0,Y 312.509,Z 230.556,A -85,B 0,C 180,E1 -15513.69,E2 -15513.69} C_VEL
LIN {X 0,Y 312.504,Z 230.553,A -85,B 0,C 180,E1 -15517.389,E2 -15517.389} C_VEL
LIN {X 0,Y 312.481,Z 230.549,A -85,B 0,C 180,E1 -15520.711,E2 -15520.711} C_VEL
LIN {X 0,Y 312.445,Z 230.568,A -85,B 0,C 180,E1 -15524.211,E2 -15524.211} C_VEL
LIN {X 0,Y 312.45,Z 230.564,A -85,B 0,C 180,E1 -15527.926,E2 -15527.926} C_VEL
LIN {X 0,Y 312.473,Z 230.564,A -85,B 0,C 180,E1 -15531.926,E2 -15531.926} C_VEL
LIN {X 0,Y 312.537,Z 230.615,A -85,B 0,C 180,E1 -15533.738,E2 -15533.738} C_VEL
LIN {X 0,Y 315.012,Z 239.939,A -85,B 0,C 180,E1 -15536.867,E2 -15536.867} C_VEL
LIN {X 0,Y 317.345,Z 250.17,A -85,B 0,C 180,E1 -15540.068,E2 -15540.068} C_VEL
LIN {X 0,Y 318.933,Z 258.34,A -85,B 0,C 180,E1 -15542.458,E2 -15542.458} C_VEL
LIN {X 0,Y 321.345,Z 267.647,A -85,B 0,C 180,E1 -15542.968,E2 -15542.968} C_VEL
LIN {X 0,Y 326.258,Z 292.641,A -85,B 0,C 180,E1 -15544.126,E2 -15544.126} C_VEL
LIN {X 0,Y 327.92,Z 304.458,A -85,B 0,C 180,E1 -15544.591,E2 -15544.591} C_VEL
LIN {X 0,Y 326.12,Z 367.933,A -85,B 0,C 180,E1 -15546.041,E2 -15546.041} C_VEL
LIN {X 0,Y 325.045,Z 381.643,A -85,B 0,C 180,E1 -15546.591,E2 -15546.591} C_VEL
LIN {X 0,Y 323.697,Z 393.995,A -85,B 0,C 180,E1 -15547.332,E2 -15547.332} C_VEL
LIN {X 0,Y 322.151,Z 405.061,A -85,B 0,C 180,E1 -15548.231,E2 -15548.231} C_VEL
LIN {X 0,Y 320.254,Z 416.599,A -85,B 0,C 180,E1 -15549.444,E2 -15549.444} C_VEL
LIN {X 0,Y 318.419,Z 427.006,A -85,B 0,C 180,E1 -15550.833,E2 -15550.833} C_VEL
LIN {X 0,Y 316.824,Z 435.54,A -85,B 0,C 180,E1 -15552.241,E2 -15552.241} C_VEL
LIN {X 0,Y 315.251,Z 443.581,A -85,B 0,C 180,E1 -15553.852,E2 -15553.852} C_VEL
LIN {X 0,Y 313.819,Z 451.191,A -85,B 0,C 180,E1 -15555.738,E2 -15555.738} C_VEL
LIN {X 0,Y 312.517,Z 457.438,A -85,B 0,C 180,E1 -15557.663,E2 -15557.663} C_VEL
LIN {X 0,Y 311.681,Z 462.436,A -85,B 0,C 180,E1 -15559.606,E2 -15559.606} C_VEL
LIN {X 0,Y 311.122,Z 466.326,A -85,B 0,C 180,E1 -15561.555,E2 -15561.555} C_VEL
LIN {X 0,Y 310.817,Z 469.211,A -85,B 0,C 180,E1 -15563.507,E2 -15563.507} C_VEL
LIN {X 0,Y 310.744,Z 471.581,A -85,B 0,C 180,E1 -15566.108,E2 -15566.108} C_VEL
LIN {X 0,Y 310.734,Z 472.183,A -85,B 0,C 180,E1 -15567.405,E2 -15567.405} C_VEL
LIN {X 0,Y 310.774,Z 472.365,A -85,B 0,C 180,E1 -15568.702,E2 -15568.702} C_VEL
LIN {X 0,Y 310.861,Z 472.137,A -85,B 0,C 180,E1 -15569.998,E2 -15569.998} C_VEL
LIN {X 0,Y 310.816,Z 471.511,A -85,B 0,C 180,E1 -15571.293,E2 -15571.293} C_VEL
LIN {X 0,Y 310.766,Z 470.489,A -85,B 0,C 180,E1 -15572.59,E2 -15572.59} C_VEL
LIN {X 0,Y 310.827,Z 469.033,A -85,B 0,C 180,E1 -15573.887,E2 -15573.887} C_VEL
LIN {X 0,Y 310.814,Z 466.12,A -85,B 0,C 180,E1 -15575.779,E2 -15575.779} C_VEL
LIN {X 0,Y 310.986,Z 461.916,A -85,B 0,C 180,E1 -15577.79,E2 -15577.79} C_VEL
LIN {X 0,Y 311.411,Z 455.602,A -85,B 0,C 180,E1 -15580.07,E2 -15580.07} C_VEL
LIN {X 0,Y 312.027,Z 448.712,A -85,B 0,C 180,E1 -15582.022,E2 -15582.022} C_VEL
LIN {X 0,Y 312.832,Z 441.678,A -85,B 0,C 180,E1 -15583.641,E2 -15583.641} C_VEL
LIN {X 0,Y 313.837,Z 433.195,A -85,B 0,C 180,E1 -15585.252,E2 -15585.252} C_VEL
LIN {X 0,Y 314.974,Z 422.697,A -85,B 0,C 180,E1 -15586.858,E2 -15586.858} C_VEL
LIN {X 0,Y 316.023,Z 412.285,A -85,B 0,C 180,E1 -15588.136,E2 -15588.136} C_VEL
LIN {X 0,Y 317.241,Z 400.913,A -85,B 0,C 180,E1 -15589.236,E2 -15589.236} C_VEL
LIN {X 0,Y 318.268,Z 389.315,A -85,B 0,C 180,E1 -15590.095,E2 -15590.095} C_VEL
LIN {X 0,Y 319.161,Z 375.978,A -85,B 0,C 180,E1 -15590.794,E2 -15590.794} C_VEL
LIN {X 0,Y 319.693,Z 363.009,A -85,B 0,C 180,E1 -15591.221,E2 -15591.221} C_VEL
LIN {X 0,Y 320.863,Z 301.589,A -85,B 0,C 180,E1 -15592.592,E2 -15592.592} C_VEL
LIN {X 0,Y 315.388,Z 259.252,A -85,B 0,C 180,E1 -15593.953,E2 -15593.953} C_VEL
LIN {X 0,Y 316.301,Z 249.484,A -85,B 0,C 180,E1 -15596.379,E2 -15596.379} C_VEL
LIN {X 0,Y 314.407,Z 239.48,A -85,B 0,C 180,E1 -15599.082,E2 -15599.082} C_VEL
LIN {X 0,Y 312.5,Z 230.559,A -85,B 0,C 180,E1 -15601.638,E2 -15601.638} C_VEL
LIN {X 0,Y 312.491,Z 230.562,A -85,B 0,C 180,E1 -15604.206,E2 -15604.206} C_VEL
LIN {X 0,Y 312.517,Z 230.559,A -85,B 0,C 180,E1 -15608.085,E2 -15608.085} C_VEL
LIN {X 0,Y 312.466,Z 230.564,A -85,B 0,C 180,E1 -15612.077,E2 -15612.077} C_VEL
LIN {X 0,Y 312.507,Z 230.559,A -85,B 0,C 180,E1 -15616.017,E2 -15616.017} C_VEL
LIN {X 0,Y 312.504,Z 230.559,A -85,B 0,C 180,E1 -15619.865,E2 -15619.865} C_VEL
LIN {X 0,Y 312.512,Z 230.554,A -85,B 0,C 180,E1 -15622.612,E2 -15622.612} C_VEL
LIN {X 0,Y 312.49,Z 230.557,A -85,B 0,C 180,E1 -15626.307,E2 -15626.307} C_VEL
LIN {X 0,Y 312.512,Z 230.554,A -85,B 0,C 180,E1 -15630.346,E2 -15630.346} C_VEL
LIN {X 0,Y 312.569,Z 230.548,A -85,B 0,C 180,E1 -15634.061,E2 -15634.061} C_VEL
LIN {X 0,Y 312.558,Z 230.554,A -85,B 0,C 180,E1 -15637.526,E2 -15637.526} C_VEL
LIN {X 0,Y 312.601,Z 230.545,A -85,B 0,C 180,E1 -15641.654,E2 -15641.654} C_VEL
LIN {X 0,Y 312.653,Z 230.539,A -85,B 0,C 180,E1 -15645.684,E2 -15645.684} C_VEL
LIN {X 0,Y 312.662,Z 230.537,A -85,B 0,C 180,E1 -15649.64,E2 -15649.64} C_VEL
LIN {X 0,Y 312.833,Z 230.514,A -85,B 0,C 180,E1 -15652.253,E2 -15652.253} C_VEL
LIN {X 0,Y 312.677,Z 230.535,A -85,B 0,C 180,E1 -15654.841,E2 -15654.841} C_VEL
LIN {X 0,Y 312.947,Z 230.496,A -85,B 0,C 180,E1 -15658.713,E2 -15658.713} C_VEL
LIN {X 0,Y 312.946,Z 230.499,A -85,B 0,C 180,E1 -15661.286,E2 -15661.286} C_VEL
LIN {X 0,Y 312.667,Z 230.538,A -85,B 0,C 180,E1 -15665.158,E2 -15665.158} C_VEL
LIN {X 0,Y 312.801,Z 230.518,A -85,B 0,C 180,E1 -15667.747,E2 -15667.747} C_VEL
LIN {X 0,Y 312.627,Z 230.538,A -85,B 0,C 180,E1 -15671.672,E2 -15671.672} C_VEL
LIN {X 0,Y 312.627,Z 230.545,A -85,B 0,C 180,E1 -15674.865,E2 -15674.865} C_VEL
LIN {X 0,Y 312.508,Z 230.554,A -85,B 0,C 180,E1 -15679.194,E2 -15679.194} C_VEL
LIN {X 0,Y 312.488,Z 230.562,A -85,B 0,C 180,E1 -15682.782,E2 -15682.782} C_VEL
LIN {X 0,Y 312.548,Z 230.549,A -85,B 0,C 180,E1 -15685.931,E2 -15685.931} C_VEL
LIN {X 0,Y 312.47,Z 230.553,A -85,B 0,C 180,E1 -15689.657,E2 -15689.657} C_VEL
LIN {X 0,Y 312.487,Z 230.554,A -85,B 0,C 180,E1 -15693.692,E2 -15693.692} C_VEL
LIN {X 0,Y 312.494,Z 230.556,A -85,B 0,C 180,E1 -15697.389,E2 -15697.389} C_VEL
LIN {X 0,Y 312.461,Z 230.56,A -85,B 0,C 180,E1 -15700.713,E2 -15700.713} C_VEL
LIN {X 0,Y 312.425,Z 230.564,A -85,B 0,C 180,E1 -15704.214,E2 -15704.214} C_VEL
LIN {X 0,Y 312.46,Z 230.563,A -85,B 0,C 180,E1 -15707.923,E2 -15707.923} C_VEL
LIN {X 0,Y 312.477,Z 230.557,A -85,B 0,C 180,E1 -15710.975,E2 -15710.975} C_VEL
LIN {X 0,Y 312.512,Z 230.558,A -85,B 0,C 180,E1 -15714.224,E2 -15714.224} C_VEL
LIN {X 0,Y 312.487,Z 230.558,A -85,B 0,C 180,E1 -15717.338,E2 -15717.338} C_VEL
LIN {X 0,Y 312.529,Z 230.552,A -85,B 0,C 180,E1 -15721.283,E2 -15721.283} C_VEL
LIN {X 0,Y 312.572,Z 230.547,A -85,B 0,C 180,E1 -15724.715,E2 -15724.715} C_VEL
LIN {X 0,Y 312.553,Z 230.551,A -85,B 0,C 180,E1 -15727.531,E2 -15727.531} C_VEL
LIN {X 0,Y 312.558,Z 230.553,A -85,B 0,C 180,E1 -15731.656,E2 -15731.656} C_VEL
LIN {X 0,Y 312.68,Z 230.54,A -85,B 0,C 180,E1 -15735.689,E2 -15735.689} C_VEL
LIN {X 0,Y 312.693,Z 230.537,A -85,B 0,C 180,E1 -15739.645,E2 -15739.645} C_VEL
LIN {X 0,Y 312.742,Z 230.66,A -85,B 0,C 180,E1 -15740.39,E2 -15740.39} C_VEL
LIN {X 0,Y 313.255,Z 232.897,A -85,B 0,C 180,E1 -15741.034,E2 -15741.034} C_VEL
LIN {X 0,Y 320.113,Z 253.198,A -85,B 0,C 180,E1 -15741.957,E2 -15741.957} C_VEL
LIN {X 0,Y 321.622,Z 261.022,A -85,B 0,C 180,E1 -15742.233,E2 -15742.233} C_VEL
LIN {X 0,Y 319.847,Z 340.126,A -85,B 0,C 180,E1 -15744.012,E2 -15744.012} C_VEL
LIN {X 0,Y 319.345,Z 353.22,A -85,B 0,C 180,E1 -15744.557,E2 -15744.557} C_VEL
LIN {X 0,Y 318.546,Z 365.905,A -85,B 0,C 180,E1 -15745.336,E2 -15745.336} C_VEL
LIN {X 0,Y 317.651,Z 377.793,A -85,B 0,C 180,E1 -15746.338,E2 -15746.338} C_VEL
LIN {X 0,Y 316.525,Z 389.689,A -85,B 0,C 180,E1 -15747.644,E2 -15747.644} C_VEL
LIN {X 0,Y 315.402,Z 399.84,A -85,B 0,C 180,E1 -15749.045,E2 -15749.045} C_VEL
LIN {X 0,Y 314.278,Z 409.164,A -85,B 0,C 180,E1 -15750.643,E2 -15750.643} C_VEL
LIN {X 0,Y 313.182,Z 418.193,A -85,B 0,C 180,E1 -15752.574,E2 -15752.574} C_VEL
LIN {X 0,Y 312.348,Z 425.465,A -85,B 0,C 180,E1 -15754.519,E2 -15754.519} C_VEL
LIN {X 0,Y 311.778,Z 431.265,A -85,B 0,C 180,E1 -15756.473,E2 -15756.473} C_VEL
LIN {X 0,Y 311.294,Z 435.84,A -85,B 0,C 180,E1 -15758.44,E2 -15758.44} C_VEL
LIN {X 0,Y 310.943,Z 439.323,A -85,B 0,C 180,E1 -15760.419,E2 -15760.419} C_VEL
LIN {X 0,Y 310.814,Z 441.051,A -85,B 0,C 180,E1 -15761.743,E2 -15761.743} C_VEL
LIN {X 0,Y 310.719,Z 442.684,A -85,B 0,C 180,E1 -15763.447,E2 -15763.447} C_VEL
LIN {X 0,Y 310.649,Z 443.748,A -85,B 0,C 180,E1 -15765.753,E2 -15765.753} C_VEL
LIN {X 0,Y 310.877,Z 443.499,A -85,B 0,C 180,E1 -15768.289,E2 -15768.289} C_VEL
LIN {X 0,Y 311.103,Z 442.648,A -85,B 0,C 180,E1 -15769.808,E2 -15769.808} C_VEL
LIN {X 0,Y 311.431,Z 441.393,A -85,B 0,C 180,E1 -15771.166,E2 -15771.166} C_VEL
LIN {X 0,Y 312.11,Z 438.67,A -85,B 0,C 180,E1 -15773.208,E2 -15773.208} C_VEL
LIN {X 0,Y 312.941,Z 434.827,A -85,B 0,C 180,E1 -15775.258,E2 -15775.258} C_VEL
LIN {X 0,Y 314.094,Z 429.74,A -85,B 0,C 180,E1 -15777.303,E2 -15777.303} C_VEL
LIN {X 0,Y 315.519,Z 423.235,A -85,B 0,C 180,E1 -15779.343,E2 -15779.343} C_VEL
LIN {X 0,Y 317.244,Z 414.933,A -85,B 0,C 180,E1 -15781.372,E2 -15781.372} C_VEL
